LIN {X 0,Y 297.37,Z 514.484,A -85,B 0,C 180,E1 -16463.214,E2 -16463.214} C_VEL
LIN {X 0,Y 296.917,Z 516.954,A -85,B 0,C 180,E1 -16465.928,E2 -16465.928} C_VEL
LIN {X 0,Y 296.729,Z 518.18,A -85,B 0,C 180,E1 -16468.643,E2 -16468.643} C_VEL
LIN {X 0,Y 296.728,Z 518.204,A -85,B 0,C 180,E1 -16471.357,E2 -16471.357} C_VEL
LIN {X 0,Y 296.915,Z 517.029,A -85,B 0,C 180,E1 -16474.072,E2 -16474.072} C_VEL
LIN {X 0,Y 297.37,Z 514.612,A -85,B 0,C 180,E1 -16476.787,E2 -16476.787} C_VEL
LIN {X 0,Y 298.048,Z 510.874,A -85,B 0,C 180,E1 -16479.501,E2 -16479.501} C_VEL
LIN {X 0,Y 299.173,Z 505.674,A -85,B 0,C 180,E1 -16482.206,E2 -16482.206} C_VEL
LIN {X 0,Y 300.7,Z 498.834,A -85,B 0,C 180,E1 -16484.898,E2 -16484.898} C_VEL
LIN {X 0,Y 302.63,Z 491.286,A -85,B 0,C 180,E1 -16487.223,E2 -16487.223} C_VEL
LIN {X 0,Y 304.325,Z 483.451,A -85,B 0,C 180,E1 -16489.214,E2 -16489.214} C_VEL
LIN {X 0,Y 306.549,Z 474.009,A -85,B 0,C 180,E1 -16491.167,E2 -16491.167} C_VEL
LIN {X 0,Y 308.714,Z 463.565,A -85,B 0,C 180,E1 -16492.946,E2 -16492.946} C_VEL
LIN {X 0,Y 311.058,Z 452.04,A -85,B 0,C 180,E1 -16494.53,E2 -16494.53} C_VEL
LIN {X 0,Y 313.15,Z 439.163,A -85,B 0,C 180,E1 -16495.967,E2 -16495.967} C_VEL
LIN {X 0,Y 313.842,Z 434.12,A -85,B 0,C 180,E1 -16496.449,E2 -16496.449} C_VEL
LIN {X 0,Y 312.158,Z 424.12,A -85,B 0,C 180,E1 -16497.579,E2 -16497.579} C_VEL
LIN {X 0,Y 309.028,Z 411.527,A -85,B 0,C 180,E1 -16498.885,E2 -16498.885} C_VEL
LIN {X 0,Y 305.023,Z 398.954,A -85,B 0,C 180,E1 -16500.071,E2 -16500.071} C_VEL
LIN {X 0,Y 300.09,Z 386.492,A -85,B 0,C 180,E1 -16501.166,E2 -16501.166} C_VEL
LIN {X 0,Y 298.999,Z 383.235,A -85,B 0,C 180,E1 -16501.435,E2 -16501.435} C_VEL
LIN {X 0,Y 299.406,Z 379.396,A -85,B 0,C 180,E1 -16504.758,E2 -16504.758} C_VEL
LIN {X 0,Y 299.702,Z 376.329,A -85,B 0,C 180,E1 -16507.568,E2 -16507.568} C_VEL
LIN {X 0,Y 299.78,Z 374.508,A -85,B 0,C 180,E1 -16509.317,E2 -16509.317} C_VEL
LIN {X 0,Y 299.694,Z 372.408,A -85,B 0,C 180,E1 -16511.373,E2 -16511.373} C_VEL
LIN {X 0,Y 299.198,Z 368.796,A -85,B 0,C 180,E1 -16515.196,E2 -16515.196} C_VEL
LIN {X 0,Y 298.695,Z 365.599,A -85,B 0,C 180,E1 -16518.845,E2 -16518.845} C_VEL
LIN {X 0,Y 298.437,Z 363.932,A -85,B 0,C 180,E1 -16520.999,E2 -16520.999} C_VEL
LIN {X 0,Y 298.422,Z 363.937,A -85,B 0,C 180,E1 -16523.93,E2 -16523.93} C_VEL
LIN {X 0,Y 298.399,Z 363.939,A -85,B 0,C 180,E1 -16527.983,E2 -16527.983} C_VEL
LIN {X 0,Y 298.468,Z 363.93,A -85,B 0,C 180,E1 -16531.904,E2 -16531.904} C_VEL
LIN {X 0,Y 298.49,Z 363.929,A -85,B 0,C 180,E1 -16534.924,E2 -16534.924} C_VEL
LIN {X 0,Y 298.454,Z 363.928,A -85,B 0,C 180,E1 -16539.315,E2 -16539.315} C_VEL
LIN {X 0,Y 298.542,Z 363.918,A -85,B 0,C 180,E1 -16542.179,E2 -16542.179} C_VEL
LIN {X 0,Y 298.59,Z 363.912,A -85,B 0,C 180,E1 -16544.574,E2 -16544.574} C_VEL
LIN {X 0,Y 297.982,Z 363.99,A -85,B 0,C 180,E1 -16545.699,E2 -16545.699} C_VEL
LIN {X 0,Y 295.123,Z 364.351,A -85,B 0,C 180,E1 -16547.531,E2 -16547.531} C_VEL
LIN {X 0,Y 292.696,Z 364.654,A -85,B 0,C 180,E1 -16549.017,E2 -16549.017} C_VEL
LIN {X 0,Y 291.706,Z 364.774,A -85,B 0,C 180,E1 -16550.17,E2 -16550.17} C_VEL
LIN {X 0,Y 291.656,Z 364.777,A -85,B 0,C 180,E1 -16550.56,E2 -16550.56} C_VEL
LIN {X 0,Y 291.752,Z 364.769,A -85,B 0,C 180,E1 -16553.082,E2 -16553.082} C_VEL
LIN {X 0,Y 291.893,Z 364.745,A -85,B 0,C 180,E1 -16558.62,E2 -16558.62} C_VEL
LIN {X 0,Y 291.893,Z 364.745,A -85,B 0,C 180,E1 -16561.379,E2 -16561.379} C_VEL
LIN {X 0,Y 291.727,Z 364.771,A -85,B 0,C 180,E1 -16566.918,E2 -16566.918} C_VEL
LIN {X 0,Y 291.577,Z 364.793,A -85,B 0,C 180,E1 -16569.713,E2 -16569.713} C_VEL
LIN {X 0,Y 291.527,Z 364.795,A -85,B 0,C 180,E1 -16573.95,E2 -16573.95} C_VEL
LIN {X 0,Y 291.491,Z 364.802,A -85,B 0,C 180,E1 -16576.817,E2 -16576.817} C_VEL
LIN {X 0,Y 291.454,Z 364.806,A -85,B 0,C 180,E1 -16579.874,E2 -16579.874} C_VEL
LIN {X 0,Y 291.404,Z 364.815,A -85,B 0,C 180,E1 -16584.205,E2 -16584.205} C_VEL
LIN {X 0,Y 291.426,Z 364.81,A -85,B 0,C 180,E1 -16587.271,E2 -16587.271} C_VEL
LIN {X 0,Y 291.341,Z 364.818,A -85,B 0,C 180,E1 -16590.436,E2 -16590.436} C_VEL
LIN {X 0,Y 291.371,Z 364.967,A -85,B 0,C 180,E1 -16592.63,E2 -16592.63} C_VEL
LIN {X 0,Y 291.946,Z 367.659,A -85,B 0,C 180,E1 -16595.292,E2 -16595.292} C_VEL
LIN {X 0,Y 292.639,Z 371.276,A -85,B 0,C 180,E1 -16598.639,E2 -16598.639} C_VEL
LIN {X 0,Y 293.493,Z 375.469,A -85,B 0,C 180,E1 -16602.105,E2 -16602.105} C_VEL
LIN {X 0,Y 294.53,Z 380.83,A -85,B 0,C 180,E1 -16606.211,E2 -16606.211} C_VEL
LIN {X 0,Y 295.49,Z 386.215,A -85,B 0,C 180,E1 -16610.045,E2 -16610.045} C_VEL
LIN {X 0,Y 296.115,Z 390.267,A -85,B 0,C 180,E1 -16612.755,E2 -16612.755} C_VEL
LIN {X 0,Y 295.651,Z 393.125,A -85,B 0,C 180,E1 -16614.523,E2 -16614.523} C_VEL
LIN {X 0,Y 295.257,Z 394.696,A -85,B 0,C 180,E1 -16615.467,E2 -16615.467} C_VEL
LIN {X 0,Y 298.115,Z 404.031,A -85,B 0,C 180,E1 -16616.148,E2 -16616.148} C_VEL
LIN {X 0,Y 302.094,Z 419.344,A -85,B 0,C 180,E1 -16617.377,E2 -16617.377} C_VEL
LIN {X 0,Y 304.904,Z 434.204,A -85,B 0,C 180,E1 -16618.725,E2 -16618.725} C_VEL
LIN {X 0,Y 306.458,Z 447.084,A -85,B 0,C 180,E1 -16620.039,E2 -16620.039} C_VEL
LIN {X 0,Y 306.776,Z 452.763,A -85,B 0,C 180,E1 -16620.66,E2 -16620.66} C_VEL
LIN {X 0,Y 304.582,Z 465.397,A -85,B 0,C 180,E1 -16621.956,E2 -16621.956} C_VEL
LIN {X 0,Y 301.948,Z 478.242,A -85,B 0,C 180,E1 -16623.567,E2 -16623.567} C_VEL
LIN {X 0,Y 299.907,Z 488.037,A -85,B 0,C 180,E1 -16625.051,E2 -16625.051} C_VEL
LIN {X 0,Y 297.566,Z 498.682,A -85,B 0,C 180,E1 -16626.964,E2 -16626.964} C_VEL
LIN {X 0,Y 295.508,Z 508.524,A -85,B 0,C 180,E1 -16629.099,E2 -16629.099} C_VEL
LIN {X 0,Y 293.411,Z 517.704,A -85,B 0,C 180,E1 -16631.495,E2 -16631.495} C_VEL
LIN {X 0,Y 291.882,Z 525.537,A -85,B 0,C 180,E1 -16633.996,E2 -16633.996} C_VEL
LIN {X 0,Y 290.679,Z 532.426,A -85,B 0,C 180,E1 -16636.721,E2 -16636.721} C_VEL
LIN {X 0,Y 289.903,Z 537.976,A -85,B 0,C 180,E1 -16639.524,E2 -16639.524} C_VEL
LIN {X 0,Y 289.637,Z 541.184,A -85,B 0,C 180,E1 -16641.628,E2 -16641.628} C_VEL
LIN {X 0,Y 289.515,Z 544.352,A -85,B 0,C 180,E1 -16644.428,E2 -16644.428} C_VEL
LIN {X 0,Y 289.519,Z 546.244,A -85,B 0,C 180,E1 -16647.217,E2 -16647.217} C_VEL
LIN {X 0,Y 289.58,Z 546.886,A -85,B 0,C 180,E1 -16650,E2 -16650} C_VEL
LIN {X 0,Y 289.522,Z 546.235,A -85,B 0,C 180,E1 -16652.783,E2 -16652.783} C_VEL
LIN {X 0,Y 289.55,Z 544.272,A -85,B 0,C 180,E1 -16655.642,E2 -16655.642} C_VEL
LIN {X 0,Y 289.637,Z 541.156,A -85,B 0,C 180,E1 -16658.371,E2 -16658.371} C_VEL
LIN {X 0,Y 290.02,Z 536.65,A -85,B 0,C 180,E1 -16661.178,E2 -16661.178} C_VEL
LIN {X 0,Y 290.906,Z 530.713,A -85,B 0,C 180,E1 -16663.98,E2 -16663.98} C_VEL
LIN {X 0,Y 292.297,Z 523.193,A -85,B 0,C 180,E1 -16666.77,E2 -16666.77} C_VEL
LIN {X 0,Y 293.903,Z 515.126,A -85,B 0,C 180,E1 -16669.196,E2 -16669.196} C_VEL
LIN {X 0,Y 296.092,Z 505.429,A -85,B 0,C 180,E1 -16671.587,E2 -16671.587} C_VEL
LIN {X 0,Y 298.214,Z 495.509,A -85,B 0,C 180,E1 -16673.618,E2 -16673.618} C_VEL
LIN {X 0,Y 300.741,Z 483.712,A -85,B 0,C 180,E1 -16675.615,E2 -16675.615} C_VEL
LIN {X 0,Y 303.171,Z 471.961,A -85,B 0,C 180,E1 -16677.248,E2 -16677.248} C_VEL
LIN {X 0,Y 305.675,Z 459.264,A -85,B 0,C 180,E1 -16678.682,E2 -16678.682} C_VEL
LIN {X 0,Y 306.763,Z 451.271,A -85,B 0,C 180,E1 -16679.474,E2 -16679.474} C_VEL
LIN {X 0,Y 305.283,Z 437.149,A -85,B 0,C 180,E1 -16680.959,E2 -16680.959} C_VEL
LIN {X 0,Y 302.891,Z 423.088,A -85,B 0,C 180,E1 -16682.264,E2 -16682.264} C_VEL
LIN {X 0,Y 299.26,Z 408.308,A -85,B 0,C 180,E1 -16683.495,E2 -16683.495} C_VEL
LIN {X 0,Y 295.225,Z 394.702,A -85,B 0,C 180,E1 -16684.5,E2 -16684.5} C_VEL
LIN {X 0,Y 295.95,Z 391.521,A -85,B 0,C 180,E1 -16686.419,E2 -16686.419} C_VEL
LIN {X 0,Y 295.895,Z 388.478,A -85,B 0,C 180,E1 -16688.39,E2 -16688.39} C_VEL
LIN {X 0,Y 294.873,Z 382.73,A -85,B 0,C 180,E1 -16692.367,E2 -16692.367} C_VEL
LIN {X 0,Y 293.937,Z 377.696,A -85,B 0,C 180,E1 -16696.102,E2 -16696.102} C_VEL
LIN {X 0,Y 293.069,Z 373.272,A -85,B 0,C 180,E1 -16699.648,E2 -16699.648} C_VEL
LIN {X 0,Y 292.307,Z 369.354,A -85,B 0,C 180,E1 -16703.053,E2 -16703.053} C_VEL
LIN {X 0,Y 291.425,Z 365.233,A -85,B 0,C 180,E1 -16707.024,E2 -16707.024} C_VEL
LIN {X 0,Y 291.346,Z 364.824,A -85,B 0,C 180,E1 -16707.596,E2 -16707.596} C_VEL
LIN {X 0,Y 291.387,Z 364.819,A -85,B 0,C 180,E1 -16711.159,E2 -16711.159} C_VEL
LIN {X 0,Y 291.422,Z 364.808,A -85,B 0,C 180,E1 -16714.273,E2 -16714.273} C_VEL
LIN {X 0,Y 291.384,Z 364.814,A -85,B 0,C 180,E1 -16717.3,E2 -16717.3} C_VEL
LIN {X 0,Y 291.46,Z 364.804,A -85,B 0,C 180,E1 -16720.271,E2 -16720.271} C_VEL
LIN {X 0,Y 291.557,Z 364.786,A -85,B 0,C 180,E1 -16724.624,E2 -16724.624} C_VEL
LIN {X 0,Y 291.54,Z 364.795,A -85,B 0,C 180,E1 -16728.881,E2 -16728.881} C_VEL
LIN {X 0,Y 291.671,Z 364.78,A -85,B 0,C 180,E1 -16731.688,E2 -16731.688} C_VEL
LIN {X 0,Y 291.628,Z 364.78,A -85,B 0,C 180,E1 -16734.469,E2 -16734.469} C_VEL
LIN {X 0,Y 291.893,Z 364.752,A -85,B 0,C 180,E1 -16738.621,E2 -16738.621} C_VEL
LIN {X 0,Y 291.892,Z 364.745,A -85,B 0,C 180,E1 -16741.38,E2 -16741.38} C_VEL
LIN {X 0,Y 291.75,Z 364.765,A -85,B 0,C 180,E1 -16746.918,E2 -16746.918} C_VEL
LIN {X 0,Y 291.633,Z 364.785,A -85,B 0,C 180,E1 -16749.712,E2 -16749.712} C_VEL
LIN {X 0,Y 291.527,Z 364.794,A -85,B 0,C 180,E1 -16753.95,E2 -16753.95} C_VEL
LIN {X 0,Y 291.491,Z 364.801,A -85,B 0,C 180,E1 -16756.818,E2 -16756.818} C_VEL
LIN {X 0,Y 291.453,Z 364.808,A -85,B 0,C 180,E1 -16759.875,E2 -16759.875} C_VEL
LIN {X 0,Y 291.403,Z 364.805,A -85,B 0,C 180,E1 -16764.205,E2 -16764.205} C_VEL
LIN {X 0,Y 291.425,Z 364.804,A -85,B 0,C 180,E1 -16767.272,E2 -16767.272} C_VEL
LIN {X 0,Y 291.34,Z 364.818,A -85,B 0,C 180,E1 -16770.437,E2 -16770.437} C_VEL
LIN {X 0,Y 291.347,Z 364.819,A -85,B 0,C 180,E1 -16773.698,E2 -16773.698} C_VEL
LIN {X 0,Y 291.375,Z 364.817,A -85,B 0,C 180,E1 -16777.253,E2 -16777.253} C_VEL
LIN {X 0,Y 291.385,Z 364.97,A -85,B 0,C 180,E1 -16778.622,E2 -16778.622} C_VEL
LIN {X 0,Y 291.885,Z 368.062,A -85,B 0,C 180,E1 -16782.391,E2 -16782.391} C_VEL
LIN {X 0,Y 292.435,Z 371.328,A -85,B 0,C 180,E1 -16786.136,E2 -16786.136} C_VEL
LIN {X 0,Y 292.753,Z 374.6,A -85,B 0,C 180,E1 -16789.595,E2 -16789.595} C_VEL
LIN {X 0,Y 292.644,Z 378.189,A -85,B 0,C 180,E1 -16793.102,E2 -16793.102} C_VEL
LIN {X 0,Y 292.223,Z 381.859,A -85,B 0,C 180,E1 -16796.416,E2 -16796.416} C_VEL
LIN {X 0,Y 292.078,Z 383.466,A -85,B 0,C 180,E1 -16797.834,E2 -16797.834} C_VEL
LIN {X 0,Y 293.241,Z 386.749,A -85,B 0,C 180,E1 -16798.103,E2 -16798.103} C_VEL
LIN {X 0,Y 298.534,Z 400.073,A -85,B 0,C 180,E1 -16799.335,E2 -16799.335} C_VEL
LIN {X 0,Y 302.565,Z 412.598,A -85,B 0,C 180,E1 -16800.583,E2 -16800.583} C_VEL
LIN {X 0,Y 305.59,Z 425.125,A -85,B 0,C 180,E1 -16801.933,E2 -16801.933} C_VEL
LIN {X 0,Y 307.35,Z 434.992,A -85,B 0,C 180,E1 -16803.1,E2 -16803.1} C_VEL
LIN {X 0,Y 305.683,Z 446.293,A -85,B 0,C 180,E1 -16804.281,E2 -16804.281} C_VEL
LIN {X 0,Y 303.559,Z 457.781,A -85,B 0,C 180,E1 -16805.736,E2 -16805.736} C_VEL
LIN {X 0,Y 301.21,Z 468.343,A -85,B 0,C 180,E1 -16807.357,E2 -16807.357} C_VEL
LIN {X 0,Y 298.819,Z 478.827,A -85,B 0,C 180,E1 -16809.342,E2 -16809.342} C_VEL
LIN {X 0,Y 296.706,Z 487.48,A -85,B 0,C 180,E1 -16811.347,E2 -16811.347} C_VEL
LIN {X 0,Y 294.766,Z 495.809,A -85,B 0,C 180,E1 -16813.731,E2 -16813.731} C_VEL
LIN {X 0,Y 293.031,Z 502.541,A -85,B 0,C 180,E1 -16816.123,E2 -16816.123} C_VEL
LIN {X 0,Y 291.594,Z 508.601,A -85,B 0,C 180,E1 -16818.883,E2 -16818.883} C_VEL
LIN {X 0,Y 290.647,Z 513.109,A -85,B 0,C 180,E1 -16821.658,E2 -16821.658} C_VEL
LIN {X 0,Y 290.078,Z 516.224,A -85,B 0,C 180,E1 -16824.439,E2 -16824.439} C_VEL
LIN {X 0,Y 289.712,Z 518.065,A -85,B 0,C 180,E1 -16827.219,E2 -16827.219} C_VEL
LIN {X 0,Y 289.594,Z 518.687,A -85,B 0,C 180,E1 -16830,E2 -16830} C_VEL
LIN {X 0,Y 289.711,Z 518.113,A -85,B 0,C 180,E1 -16832.781,E2 -16832.781} C_VEL
LIN {X 0,Y 290.059,Z 516.324,A -85,B 0,C 180,E1 -16835.562,E2 -16835.562} C_VEL
LIN {X 0,Y 290.645,Z 513.261,A -85,B 0,C 180,E1 -16838.342,E2 -16838.342} C_VEL
LIN {X 0,Y 291.572,Z 508.818,A -85,B 0,C 180,E1 -16841.118,E2 -16841.118} C_VEL
LIN {X 0,Y 292.952,Z 502.829,A -85,B 0,C 180,E1 -16843.881,E2 -16843.881} C_VEL
LIN {X 0,Y 294.741,Z 496.162,A -85,B 0,C 180,E1 -16846.271,E2 -16846.271} C_VEL
LIN {X 0,Y 296.503,Z 488.39,A -85,B 0,C 180,E1 -16848.536,E2 -16848.536} C_VEL
LIN {X 0,Y 298.705,Z 479.34,A -85,B 0,C 180,E1 -16850.667,E2 -16850.667} C_VEL
LIN {X 0,Y 301.136,Z 468.954,A -85,B 0,C 180,E1 -16852.649,E2 -16852.649} C_VEL
LIN {X 0,Y 303.481,Z 458.512,A -85,B 0,C 180,E1 -16854.271,E2 -16854.271} C_VEL
LIN {X 0,Y 305.566,Z 447.194,A -85,B 0,C 180,E1 -16855.73,E2 -16855.73} C_VEL
LIN {X 0,Y 307.42,Z 435.802,A -85,B 0,C 180,E1 -16856.926,E2 -16856.926} C_VEL
LIN {X 0,Y 305.267,Z 423.348,A -85,B 0,C 180,E1 -16858.384,E2 -16858.384} C_VEL
LIN {X 0,Y 301.631,Z 409.433,A -85,B 0,C 180,E1 -16859.864,E2 -16859.864} C_VEL
LIN {X 0,Y 297.328,Z 396.7,A -85,B 0,C 180,E1 -16861.109,E2 -16861.109} C_VEL
LIN {X 0,Y 292.847,Z 385.944,A -85,B 0,C 180,E1 -16862.097,E2 -16862.097} C_VEL
LIN {X 0,Y 292.067,Z 383.454,A -85,B 0,C 180,E1 -16862.302,E2 -16862.302} C_VEL
LIN {X 0,Y 292.445,Z 380.152,A -85,B 0,C 180,E1 -16865.224,E2 -16865.224} C_VEL
LIN {X 0,Y 292.764,Z 376.571,A -85,B 0,C 180,E1 -16868.62,E2 -16868.62} C_VEL
LIN {X 0,Y 292.651,Z 373.314,A -85,B 0,C 180,E1 -16871.887,E2 -16871.887} C_VEL
LIN {X 0,Y 292.163,Z 369.759,A -85,B 0,C 180,E1 -16875.765,E2 -16875.765} C_VEL
LIN {X 0,Y 291.685,Z 366.668,A -85,B 0,C 180,E1 -16879.416,E2 -16879.416} C_VEL
LIN {X 0,Y 291.371,Z 364.813,A -85,B 0,C 180,E1 -16881.803,E2 -16881.803} C_VEL
LIN {X 0,Y 291.373,Z 364.817,A -85,B 0,C 180,E1 -16885.095,E2 -16885.095} C_VEL
LIN {X 0,Y 291.376,Z 364.814,A -85,B 0,C 180,E1 -16887.951,E2 -16887.951} C_VEL
LIN {X 0,Y 291.386,Z 364.813,A -85,B 0,C 180,E1 -16891.159,E2 -16891.159} C_VEL
LIN {X 0,Y 291.421,Z 364.806,A -85,B 0,C 180,E1 -16894.272,E2 -16894.272} C_VEL
LIN {X 0,Y 291.386,Z 364.814,A -85,B 0,C 180,E1 -16897.3,E2 -16897.3} C_VEL
LIN {X 0,Y 291.462,Z 364.806,A -85,B 0,C 180,E1 -16900.27,E2 -16900.27} C_VEL
LIN {X 0,Y 291.559,Z 364.788,A -85,B 0,C 180,E1 -16904.624,E2 -16904.624} C_VEL
LIN {X 0,Y 291.542,Z 364.791,A -85,B 0,C 180,E1 -16908.881,E2 -16908.881} C_VEL
LIN {X 0,Y 291.656,Z 364.777,A -85,B 0,C 180,E1 -16910.56,E2 -16910.56} C_VEL
LIN {X 0,Y 291.383,Z 364.809,A -85,B 0,C 180,E1 -16911.331,E2 -16911.331} C_VEL
LIN {X 0,Y 290.021,Z 364.983,A -85,B 0,C 180,E1 -16912.468,E2 -16912.468} C_VEL
LIN {X 0,Y 285.621,Z 365.529,A -85,B 0,C 180,E1 -16915.111,E2 -16915.111} C_VEL
LIN {X 0,Y 284.668,Z 365.651,A -85,B 0,C 180,E1 -16916.294,E2 -16916.294} C_VEL
LIN {X 0,Y 284.65,Z 365.649,A -85,B 0,C 180,E1 -16916.694,E2 -16916.694} C_VEL
LIN {X 0,Y 284.928,Z 365.62,A -85,B 0,C 180,E1 -16920,E2 -16920} C_VEL
LIN {X 0,Y 284.747,Z 365.641,A -85,B 0,C 180,E1 -16922.829,E2 -16922.829} C_VEL
LIN {X 0,Y 284.678,Z 365.647,A -85,B 0,C 180,E1 -16927.09,E2 -16927.09} C_VEL
LIN {X 0,Y 284.522,Z 365.671,A -85,B 0,C 180,E1 -16929.957,E2 -16929.957} C_VEL
LIN {X 0,Y 284.487,Z 365.673,A -85,B 0,C 180,E1 -16934.302,E2 -16934.302} C_VEL
LIN {X 0,Y 284.43,Z 365.681,A -85,B 0,C 180,E1 -16937.248,E2 -16937.248} C_VEL
LIN {X 0,Y 284.384,Z 365.687,A -85,B 0,C 180,E1 -16940.242,E2 -16940.242} C_VEL
LIN {X 0,Y 284.373,Z 365.692,A -85,B 0,C 180,E1 -16943.875,E2 -16943.875} C_VEL
LIN {X 0,Y 284.4,Z 365.685,A -85,B 0,C 180,E1 -16947.173,E2 -16947.173} C_VEL
LIN {X 0,Y 284.299,Z 365.7,A -85,B 0,C 180,E1 -16951.274,E2 -16951.274} C_VEL
LIN {X 0,Y 284.976,Z 368.813,A -85,B 0,C 180,E1 -16954.556,E2 -16954.556} C_VEL
LIN {X 0,Y 285.691,Z 372.513,A -85,B 0,C 180,E1 -16958.075,E2 -16958.075} C_VEL
LIN {X 0,Y 286.476,Z 376.426,A -85,B 0,C 180,E1 -16961.481,E2 -16961.481} C_VEL
LIN {X 0,Y 287.348,Z 381.061,A -85,B 0,C 180,E1 -16965.177,E2 -16965.177} C_VEL
LIN {X 0,Y 288.301,Z 386.346,A -85,B 0,C 180,E1 -16969.086,E2 -16969.086} C_VEL
LIN {X 0,Y 289.102,Z 391.33,A -85,B 0,C 180,E1 -16972.573,E2 -16972.573} C_VEL
LIN {X 0,Y 288.719,Z 393.944,A -85,B 0,C 180,E1 -16974.252,E2 -16974.252} C_VEL
LIN {X 0,Y 288.568,Z 394.496,A -85,B 0,C 180,E1 -16974.592,E2 -16974.592} C_VEL
LIN {X 0,Y 291.432,Z 403.799,A -85,B 0,C 180,E1 -16975.305,E2 -16975.305} C_VEL
LIN {X 0,Y 295.43,Z 418.879,A -85,B 0,C 180,E1 -16976.571,E2 -16976.571} C_VEL
LIN {X 0,Y 298.17,Z 432.949,A -85,B 0,C 180,E1 -16977.893,E2 -16977.893} C_VEL
LIN {X 0,Y 299.659,Z 444.735,A -85,B 0,C 180,E1 -16979.117,E2 -16979.117} C_VEL
LIN {X 0,Y 300.331,Z 453.325,A -85,B 0,C 180,E1 -16980.086,E2 -16980.086} C_VEL
LIN {X 0,Y 298.011,Z 466.352,A -85,B 0,C 180,E1 -16981.474,E2 -16981.474} C_VEL
LIN {X 0,Y 295.292,Z 478.986,A -85,B 0,C 180,E1 -16983.114,E2 -16983.114} C_VEL
LIN {X 0,Y 292.964,Z 489.599,A -85,B 0,C 180,E1 -16984.798,E2 -16984.798} C_VEL
LIN {X 0,Y 290.514,Z 500.257,A -85,B 0,C 180,E1 -16986.821,E2 -16986.821} C_VEL
LIN {X 0,Y 288.159,Z 510.909,A -85,B 0,C 180,E1 -16989.289,E2 -16989.289} C_VEL
LIN {X 0,Y 286.088,Z 519.627,A -85,B 0,C 180,E1 -16991.747,E2 -16991.747} C_VEL
LIN {X 0,Y 284.566,Z 527.296,A -85,B 0,C 180,E1 -16994.405,E2 -16994.405} C_VEL
LIN {X 0,Y 283.457,Z 533.558,A -85,B 0,C 180,E1 -16997.106,E2 -16997.106} C_VEL
LIN {X 0,Y 282.725,Z 538.754,A -85,B 0,C 180,E1 -16999.979,E2 -16999.979} C_VEL
LIN {X 0,Y 282.466,Z 542.582,A -85,B 0,C 180,E1 -17002.853,E2 -17002.853} C_VEL
LIN {X 0,Y 282.411,Z 545.109,A -85,B 0,C 180,E1 -17005.718,E2 -17005.718} C_VEL
LIN {X 0,Y 282.446,Z 546.378,A -85,B 0,C 180,E1 -17008.574,E2 -17008.574} C_VEL
LIN {X 0,Y 282.493,Z 546.541,A -85,B 0,C 180,E1 -17010,E2 -17010} C_VEL
LIN {X 0,Y 282.448,Z 545.89,A -85,B 0,C 180,E1 -17012.852,E2 -17012.852} C_VEL
LIN {X 0,Y 282.463,Z 543.984,A -85,B 0,C 180,E1 -17015.712,E2 -17015.712} C_VEL
LIN {X 0,Y 282.575,Z 540.805,A -85,B 0,C 180,E1 -17018.582,E2 -17018.582} C_VEL
LIN {X 0,Y 282.987,Z 536.295,A -85,B 0,C 180,E1 -17021.46,E2 -17021.46} C_VEL
LIN {X 0,Y 283.944,Z 530.354,A -85,B 0,C 180,E1 -17024.33,E2 -17024.33} C_VEL
LIN {X 0,Y 285.422,Z 522.828,A -85,B 0,C 180,E1 -17027.186,E2 -17027.186} C_VEL
LIN {X 0,Y 287.112,Z 514.751,A -85,B 0,C 180,E1 -17029.668,E2 -17029.668} C_VEL
LIN {X 0,Y 289.394,Z 505.041,A -85,B 0,C 180,E1 -17032.112,E2 -17032.112} C_VEL
LIN {X 0,Y 291.639,Z 495.106,A -85,B 0,C 180,E1 -17034.184,E2 -17034.184} C_VEL
LIN {X 0,Y 294.279,Z 483.286,A -85,B 0,C 180,E1 -17036.22,E2 -17036.22} C_VEL
LIN {X 0,Y 296.797,Z 471.503,A -85,B 0,C 180,E1 -17037.883,E2 -17037.883} C_VEL
LIN {X 0,Y 299.432,Z 458.763,A -85,B 0,C 180,E1 -17039.338,E2 -17039.338} C_VEL
LIN {X 0,Y 300.265,Z 452.33,A -85,B 0,C 180,E1 -17040.001,E2 -17040.001} C_VEL
LIN {X 0,Y 298.95,Z 438.724,A -85,B 0,C 180,E1 -17041.496,E2 -17041.496} C_VEL
LIN {X 0,Y 296.619,Z 424.538,A -85,B 0,C 180,E1 -17042.883,E2 -17042.883} C_VEL
LIN {X 0,Y 293.229,Z 410.18,A -85,B 0,C 180,E1 -17044.144,E2 -17044.144} C_VEL
LIN {X 0,Y 288.548,Z 394.468,A -85,B 0,C 180,E1 -17045.393,E2 -17045.393} C_VEL
LIN {X 0,Y 289.073,Z 391.269,A -85,B 0,C 180,E1 -17047.431,E2 -17047.431} C_VEL
LIN {X 0,Y 288.499,Z 387.445,A -85,B 0,C 180,E1 -17050.08,E2 -17050.08} C_VEL
LIN {X 0,Y 287.553,Z 382.09,A -85,B 0,C 180,E1 -17053.99,E2 -17053.99} C_VEL
LIN {X 0,Y 286.737,Z 377.831,A -85,B 0,C 180,E1 -17057.334,E2 -17057.334} C_VEL
LIN {X 0,Y 286.042,Z 374.282,A -85,B 0,C 180,E1 -17060.297,E2 -17060.297} C_VEL
LIN {X 0,Y 285.15,Z 369.758,A -85,B 0,C 180,E1 -17064.424,E2 -17064.424} C_VEL
LIN {X 0,Y 284.304,Z 365.7,A -85,B 0,C 180,E1 -17068.649,E2 -17068.649} C_VEL
LIN {X 0,Y 284.401,Z 365.685,A -85,B 0,C 180,E1 -17072.826,E2 -17072.826} C_VEL
LIN {X 0,Y 284.369,Z 365.685,A -85,B 0,C 180,E1 -17076.707,E2 -17076.707} C_VEL
LIN {X 0,Y 284.406,Z 365.678,A -85,B 0,C 180,E1 -17081.262,E2 -17081.262} C_VEL
LIN {X 0,Y 284.494,Z 365.665,A -85,B 0,C 180,E1 -17084.459,E2 -17084.459} C_VEL
LIN {X 0,Y 284.491,Z 365.674,A -85,B 0,C 180,E1 -17088.602,E2 -17088.602} C_VEL
LIN {X 0,Y 284.625,Z 365.655,A -85,B 0,C 180,E1 -17091.48,E2 -17091.48} C_VEL
LIN {X 0,Y 284.597,Z 365.655,A -85,B 0,C 180,E1 -17094.331,E2 -17094.331} C_VEL
LIN {X 0,Y 284.859,Z 365.629,A -85,B 0,C 180,E1 -17098.587,E2 -17098.587} C_VEL
LIN {X 0,Y 284.858,Z 365.621,A -85,B 0,C 180,E1 -17101.414,E2 -17101.414} C_VEL
LIN {X 0,Y 284.702,Z 365.642,A -85,B 0,C 180,E1 -17107.09,E2 -17107.09} C_VEL
LIN {X 0,Y 284.57,Z 365.664,A -85,B 0,C 180,E1 -17109.955,E2 -17109.955} C_VEL
LIN {X 0,Y 284.486,Z 365.669,A -85,B 0,C 180,E1 -17114.303,E2 -17114.303} C_VEL
LIN {X 0,Y 284.429,Z 365.679,A -85,B 0,C 180,E1 -17117.248,E2 -17117.248} C_VEL
LIN {X 0,Y 284.381,Z 365.685,A -85,B 0,C 180,E1 -17120.242,E2 -17120.242} C_VEL
LIN {X 0,Y 284.372,Z 365.682,A -85,B 0,C 180,E1 -17123.876,E2 -17123.876} C_VEL
LIN {X 0,Y 284.4,Z 365.679,A -85,B 0,C 180,E1 -17127.174,E2 -17127.174} C_VEL
LIN {X 0,Y 284.299,Z 365.697,A -85,B 0,C 180,E1 -17131.274,E2 -17131.274} C_VEL
LIN {X 0,Y 284.343,Z 365.693,A -85,B 0,C 180,E1 -17135.348,E2 -17135.348} C_VEL
LIN {X 0,Y 284.359,Z 365.878,A -85,B 0,C 180,E1 -17137.731,E2 -17137.731} C_VEL
LIN {X 0,Y 284.892,Z 369.049,A -85,B 0,C 180,E1 -17141.764,E2 -17141.764} C_VEL
LIN {X 0,Y 285.405,Z 372.268,A -85,B 0,C 180,E1 -17145.571,E2 -17145.571} C_VEL
LIN {X 0,Y 285.729,Z 374.826,A -85,B 0,C 180,E1 -17148.386,E2 -17148.386} C_VEL
LIN {X 0,Y 285.793,Z 376.621,A -85,B 0,C 180,E1 -17150.255,E2 -17150.255} C_VEL
LIN {X 0,Y 285.737,Z 378.426,A -85,B 0,C 180,E1 -17152.055,E2 -17152.055} C_VEL
LIN {X 0,Y 285.332,Z 382.107,A -85,B 0,C 180,E1 -17155.492,E2 -17155.492} C_VEL
LIN {X 0,Y 285.17,Z 383.727,A -85,B 0,C 180,E1 -17156.923,E2 -17156.923} C_VEL
LIN {X 0,Y 286.3,Z 386.895,A -85,B 0,C 180,E1 -17157.186,E2 -17157.186} C_VEL
LIN {X 0,Y 291.115,Z 398.564,A -85,B 0,C 180,E1 -17158.323,E2 -17158.323} C_VEL
LIN {X 0,Y 295.605,Z 411.983,A -85,B 0,C 180,E1 -17159.714,E2 -17159.714} C_VEL
LIN {X 0,Y 298.79,Z 424.625,A -85,B 0,C 180,E1 -17161.126,E2 -17161.126} C_VEL
LIN {X 0,Y 300.967,Z 437.063,A -85,B 0,C 180,E1 -17162.652,E2 -17162.652} C_VEL
LIN {X 0,Y 298.826,Z 449.547,A -85,B 0,C 180,E1 -17164.021,E2 -17164.021} C_VEL
LIN {X 0,Y 296.325,Z 461.601,A -85,B 0,C 180,E1 -17165.664,E2 -17165.664} C_VEL
LIN {X 0,Y 294.29,Z 470.683,A -85,B 0,C 180,E1 -17167.165,E2 -17167.165} C_VEL
LIN {X 0,Y 291.803,Z 480.808,A -85,B 0,C 180,E1 -17169.191,E2 -17169.191} C_VEL
LIN {X 0,Y 289.703,Z 488.943,A -85,B 0,C 180,E1 -17171.18,E2 -17171.18} C_VEL
LIN {X 0,Y 287.671,Z 497.254,A -85,B 0,C 180,E1 -17173.683,E2 -17173.683} C_VEL
LIN {X 0,Y 286.12,Z 502.899,A -85,B 0,C 180,E1 -17175.781,E2 -17175.781} C_VEL
LIN {X 0,Y 284.618,Z 508.954,A -85,B 0,C 180,E1 -17178.607,E2 -17178.607} C_VEL
LIN {X 0,Y 283.616,Z 513.458,A -85,B 0,C 180,E1 -17181.45,E2 -17181.45} C_VEL
LIN {X 0,Y 283.019,Z 516.57,A -85,B 0,C 180,E1 -17184.3,E2 -17184.3} C_VEL
LIN {X 0,Y 282.638,Z 518.41,A -85,B 0,C 180,E1 -17187.15,E2 -17187.15} C_VEL
LIN {X 0,Y 282.508,Z 519.032,A -85,B 0,C 180,E1 -17190,E2 -17190} C_VEL
LIN {X 0,Y 282.637,Z 518.457,A -85,B 0,C 180,E1 -17192.851,E2 -17192.851} C_VEL
LIN {X 0,Y 283.003,Z 516.669,A -85,B 0,C 180,E1 -17195.701,E2 -17195.701} C_VEL
LIN {X 0,Y 283.612,Z 513.608,A -85,B 0,C 180,E1 -17198.551,E2 -17198.551} C_VEL
LIN {X 0,Y 284.599,Z 509.168,A -85,B 0,C 180,E1 -17201.394,E2 -17201.394} C_VEL
LIN {X 0,Y 286.044,Z 503.184,A -85,B 0,C 180,E1 -17204.223,E2 -17204.223} C_VEL
LIN {X 0,Y 287.937,Z 496.522,A -85,B 0,C 180,E1 -17206.666,E2 -17206.666} C_VEL
LIN {X 0,Y 289.69,Z 489.129,A -85,B 0,C 180,E1 -17208.887,E2 -17208.887} C_VEL
LIN {X 0,Y 292.095,Z 479.722,A -85,B 0,C 180,E1 -17211.156,E2 -17211.156} C_VEL
LIN {X 0,Y 294.608,Z 469.356,A -85,B 0,C 180,E1 -17213.18,E2 -17213.18} C_VEL
LIN {X 0,Y 297.035,Z 458.94,A -85,B 0,C 180,E1 -17214.833,E2 -17214.833} C_VEL
LIN {X 0,Y 299.216,Z 447.659,A -85,B 0,C 180,E1 -17216.317,E2 -17216.317} C_VEL
LIN {X 0,Y 300.993,Z 437.048,A -85,B 0,C 180,E1 -17217.466,E2 -17217.466} C_VEL
LIN {X 0,Y 298.791,Z 424.446,A -85,B 0,C 180,E1 -17219.011,E2 -17219.011} C_VEL
LIN {X 0,Y 295.515,Z 411.619,A -85,B 0,C 180,E1 -17220.445,E2 -17220.445} C_VEL
LIN {X 0,Y 290.891,Z 397.772,A -85,B 0,C 180,E1 -17221.873,E2 -17221.873} C_VEL
LIN {X 0,Y 286.329,Z 386.933,A -85,B 0,C 180,E1 -17222.935,E2 -17222.935} C_VEL
LIN {X 0,Y 285.281,Z 384.242,A -85,B 0,C 180,E1 -17223.171,E2 -17223.171} C_VEL
LIN {X 0,Y 285.177,Z 383.615,A -85,B 0,C 180,E1 -17223.247,E2 -17223.247} C_VEL
LIN {X 0,Y 285.564,Z 380.386,A -85,B 0,C 180,E1 -17226.205,E2 -17226.205} C_VEL
LIN {X 0,Y 285.751,Z 378.442,A -85,B 0,C 180,E1 -17228.09,E2 -17228.09} C_VEL
LIN {X 0,Y 285.806,Z 376.206,A -85,B 0,C 180,E1 -17230.333,E2 -17230.333} C_VEL
LIN {X 0,Y 285.494,Z 373.191,A -85,B 0,C 180,E1 -17233.574,E2 -17233.574} C_VEL
LIN {X 0,Y 284.97,Z 369.611,A -85,B 0,C 180,E1 -17237.721,E2 -17237.721} C_VEL
LIN {X 0,Y 284.688,Z 367.683,A -85,B 0,C 180,E1 -17240.069,E2 -17240.069} C_VEL
LIN {X 0,Y 284.371,Z 365.686,A -85,B 0,C 180,E1 -17242.944,E2 -17242.944} C_VEL
LIN {X 0,Y 284.312,Z 365.695,A -85,B 0,C 180,E1 -17247.19,E2 -17247.19} C_VEL
LIN {X 0,Y 284.363,Z 365.69,A -85,B 0,C 180,E1 -17250.376,E2 -17250.376} C_VEL
LIN {X 0,Y 284.382,Z 365.683,A -85,B 0,C 180,E1 -17253.587,E2 -17253.587} C_VEL
LIN {X 0,Y 284.371,Z 365.684,A -85,B 0,C 180,E1 -17256.707,E2 -17256.707} C_VEL
LIN {X 0,Y 284.408,Z 365.681,A -85,B 0,C 180,E1 -17261.262,E2 -17261.262} C_VEL
LIN {X 0,Y 284.497,Z 365.669,A -85,B 0,C 180,E1 -17264.459,E2 -17264.459} C_VEL
LIN {X 0,Y 284.493,Z 365.667,A -85,B 0,C 180,E1 -17268.601,E2 -17268.601} C_VEL
LIN {X 0,Y 284.664,Z 365.645,A -85,B 0,C 180,E1 -17271.481,E2 -17271.481} C_VEL
LIN {X 0,Y 284.606,Z 365.653,A -85,B 0,C 180,E1 -17274.331,E2 -17274.331} C_VEL
LIN {X 0,Y 284.65,Z 365.649,A -85,B 0,C 180,E1 -17276.694,E2 -17276.694} C_VEL
LIN {X 0,Y 284.179,Z 365.712,A -85,B 0,C 180,E1 -17277.877,E2 -17277.877} C_VEL
LIN {X 0,Y 282.734,Z 365.898,A -85,B 0,C 180,E1 -17279.04,E2 -17279.04} C_VEL
LIN {X 0,Y 278.139,Z 366.47,A -85,B 0,C 180,E1 -17282.174,E2 -17282.174} C_VEL
LIN {X 0,Y 277.682,Z 366.52,A -85,B 0,C 180,E1 -17282.994,E2 -17282.994} C_VEL
LIN {X 0,Y 277.632,Z 366.524,A -85,B 0,C 180,E1 -17287.271,E2 -17287.271} C_VEL
LIN {X 0,Y 277.465,Z 366.547,A -85,B 0,C 180,E1 -17290.213,E2 -17290.213} C_VEL
LIN {X 0,Y 277.439,Z 366.552,A -85,B 0,C 180,E1 -17294.674,E2 -17294.674} C_VEL
LIN {X 0,Y 277.35,Z 366.565,A -85,B 0,C 180,E1 -17299.233,E2 -17299.233} C_VEL
LIN {X 0,Y 277.332,Z 366.569,A -85,B 0,C 180,E1 -17303.92,E2 -17303.92} C_VEL
LIN {X 0,Y 277.329,Z 366.567,A -85,B 0,C 180,E1 -17307.505,E2 -17307.505} C_VEL
LIN {X 0,Y 277.307,Z 366.679,A -85,B 0,C 180,E1 -17310.186,E2 -17310.186} C_VEL
LIN {X 0,Y 277.941,Z 369.968,A -85,B 0,C 180,E1 -17313.799,E2 -17313.799} C_VEL
LIN {X 0,Y 278.656,Z 373.488,A -85,B 0,C 180,E1 -17317.251,E2 -17317.251} C_VEL
LIN {X 0,Y 279.49,Z 377.632,A -85,B 0,C 180,E1 -17321.029,E2 -17321.029} C_VEL
LIN {X 0,Y 280.501,Z 383.019,A -85,B 0,C 180,E1 -17325.448,E2 -17325.448} C_VEL
LIN {X 0,Y 281.466,Z 388.399,A -85,B 0,C 180,E1 -17329.518,E2 -17329.518} C_VEL
LIN {X 0,Y 282.074,Z 392.197,A -85,B 0,C 180,E1 -17332.245,E2 -17332.245} C_VEL
LIN {X 0,Y 281.914,Z 394.334,A -85,B 0,C 180,E1 -17333.678,E2 -17333.678} C_VEL
LIN {X 0,Y 283.742,Z 400.399,A -85,B 0,C 180,E1 -17334.157,E2 -17334.157} C_VEL
LIN {X 0,Y 287.649,Z 413.665,A -85,B 0,C 180,E1 -17335.301,E2 -17335.301} C_VEL
LIN {X 0,Y 290.805,Z 427.946,A -85,B 0,C 180,E1 -17336.644,E2 -17336.644} C_VEL
LIN {X 0,Y 292.921,Z 442.283,A -85,B 0,C 180,E1 -17338.14,E2 -17338.14} C_VEL
LIN {X 0,Y 293.842,Z 454.77,A -85,B 0,C 180,E1 -17339.58,E2 -17339.58} C_VEL
LIN {X 0,Y 291.148,Z 468.649,A -85,B 0,C 180,E1 -17341.133,E2 -17341.133} C_VEL
LIN {X 0,Y 288.412,Z 480.859,A -85,B 0,C 180,E1 -17342.812,E2 -17342.812} C_VEL
LIN {X 0,Y 286.002,Z 491.159,A -85,B 0,C 180,E1 -17344.53,E2 -17344.53} C_VEL
LIN {X 0,Y 283.525,Z 501.653,A -85,B 0,C 180,E1 -17346.633,E2 -17346.633} C_VEL
LIN {X 0,Y 281.454,Z 510.534,A -85,B 0,C 180,E1 -17348.772,E2 -17348.772} C_VEL
LIN {X 0,Y 279.261,Z 519.26,A -85,B 0,C 180,E1 -17351.284,E2 -17351.284} C_VEL
LIN {X 0,Y 277.72,Z 526.506,A -85,B 0,C 180,E1 -17353.837,E2 -17353.837} C_VEL
LIN {X 0,Y 276.451,Z 533.204,A -85,B 0,C 180,E1 -17356.773,E2 -17356.773} C_VEL
LIN {X 0,Y 275.682,Z 538.404,A -85,B 0,C 180,E1 -17359.72,E2 -17359.72} C_VEL
LIN {X 0,Y 275.372,Z 542.234,A -85,B 0,C 180,E1 -17362.668,E2 -17362.668} C_VEL
LIN {X 0,Y 275.317,Z 544.762,A -85,B 0,C 180,E1 -17365.608,E2 -17365.608} C_VEL
LIN {X 0,Y 275.366,Z 546.033,A -85,B 0,C 180,E1 -17368.537,E2 -17368.537} C_VEL
LIN {X 0,Y 275.409,Z 546.196,A -85,B 0,C 180,E1 -17370,E2 -17370} C_VEL
LIN {X 0,Y 275.375,Z 545.545,A -85,B 0,C 180,E1 -17372.926,E2 -17372.926} C_VEL
LIN {X 0,Y 275.379,Z 543.637,A -85,B 0,C 180,E1 -17375.859,E2 -17375.859} C_VEL
LIN {X 0,Y 275.491,Z 540.454,A -85,B 0,C 180,E1 -17378.805,E2 -17378.805} C_VEL
LIN {X 0,Y 275.968,Z 535.942,A -85,B 0,C 180,E1 -17381.755,E2 -17381.755} C_VEL
LIN {X 0,Y 276.975,Z 529.994,A -85,B 0,C 180,E1 -17384.699,E2 -17384.699} C_VEL
LIN {X 0,Y 278.558,Z 522.463,A -85,B 0,C 180,E1 -17387.623,E2 -17387.623} C_VEL
LIN {X 0,Y 280.36,Z 514.378,A -85,B 0,C 180,E1 -17390.162,E2 -17390.162} C_VEL
LIN {X 0,Y 282.749,Z 504.655,A -85,B 0,C 180,E1 -17392.66,E2 -17392.66} C_VEL
LIN {X 0,Y 285.082,Z 494.703,A -85,B 0,C 180,E1 -17394.777,E2 -17394.777} C_VEL
LIN {X 0,Y 287.862,Z 482.862,A -85,B 0,C 180,E1 -17396.851,E2 -17396.851} C_VEL
LIN {X 0,Y 290.511,Z 471.049,A -85,B 0,C 180,E1 -17398.541,E2 -17398.541} C_VEL
LIN {X 0,Y 293.21,Z 458.262,A -85,B 0,C 180,E1 -17400.024,E2 -17400.024} C_VEL
LIN {X 0,Y 293.815,Z 453.304,A -85,B 0,C 180,E1 -17400.559,E2 -17400.559} C_VEL
LIN {X 0,Y 292.556,Z 439.542,A -85,B 0,C 180,E1 -17402.135,E2 -17402.135} C_VEL
LIN {X 0,Y 290.229,Z 425.182,A -85,B 0,C 180,E1 -17403.603,E2 -17403.603} C_VEL
LIN {X 0,Y 286.774,Z 410.367,A -85,B 0,C 180,E1 -17404.961,E2 -17404.961} C_VEL
LIN {X 0,Y 282.587,Z 397.049,A -85,B 0,C 180,E1 -17406.091,E2 -17406.091} C_VEL
LIN {X 0,Y 281.853,Z 394.324,A -85,B 0,C 180,E1 -17406.296,E2 -17406.296} C_VEL
LIN {X 0,Y 282.057,Z 392.133,A -85,B 0,C 180,E1 -17407.745,E2 -17407.745} C_VEL
LIN {X 0,Y 281.226,Z 387.036,A -85,B 0,C 180,E1 -17411.434,E2 -17411.434} C_VEL
LIN {X 0,Y 280.317,Z 381.871,A -85,B 0,C 180,E1 -17415.412,E2 -17415.412} C_VEL
LIN {X 0,Y 279.437,Z 377.367,A -85,B 0,C 180,E1 -17419.163,E2 -17419.163} C_VEL
LIN {X 0,Y 278.633,Z 373.398,A -85,B 0,C 180,E1 -17422.746,E2 -17422.746} C_VEL
LIN {X 0,Y 277.853,Z 369.548,A -85,B 0,C 180,E1 -17426.585,E2 -17426.585} C_VEL
LIN {X 0,Y 277.289,Z 366.572,A -85,B 0,C 180,E1 -17429.962,E2 -17429.962} C_VEL
LIN {X 0,Y 277.363,Z 366.562,A -85,B 0,C 180,E1 -17432.865,E2 -17432.865} C_VEL
LIN {X 0,Y 277.331,Z 366.563,A -85,B 0,C 180,E1 -17436.08,E2 -17436.08} C_VEL
LIN {X 0,Y 277.347,Z 366.559,A -85,B 0,C 180,E1 -17440.767,E2 -17440.767} C_VEL
LIN {X 0,Y 277.438,Z 366.551,A -85,B 0,C 180,E1 -17445.326,E2 -17445.326} C_VEL
LIN {X 0,Y 277.463,Z 366.542,A -85,B 0,C 180,E1 -17449.787,E2 -17449.787} C_VEL
LIN {X 0,Y 277.632,Z 366.524,A -85,B 0,C 180,E1 -17452.729,E2 -17452.729} C_VEL
LIN {X 0,Y 277.825,Z 366.504,A -85,B 0,C 180,E1 -17458.551,E2 -17458.551} C_VEL
LIN {X 0,Y 277.824,Z 366.498,A -85,B 0,C 180,E1 -17461.45,E2 -17461.45} C_VEL
LIN {X 0,Y 277.657,Z 366.518,A -85,B 0,C 180,E1 -17467.271,E2 -17467.271} C_VEL
LIN {X 0,Y 277.511,Z 366.541,A -85,B 0,C 180,E1 -17470.211,E2 -17470.211} C_VEL
LIN {X 0,Y 277.439,Z 366.545,A -85,B 0,C 180,E1 -17474.674,E2 -17474.674} C_VEL
LIN {X 0,Y 277.348,Z 366.562,A -85,B 0,C 180,E1 -17479.234,E2 -17479.234} C_VEL
LIN {X 0,Y 277.322,Z 366.559,A -85,B 0,C 180,E1 -17484.171,E2 -17484.171} C_VEL
LIN {X 0,Y 277.329,Z 366.561,A -85,B 0,C 180,E1 -17487.506,E2 -17487.506} C_VEL
LIN {X 0,Y 277.274,Z 366.57,A -85,B 0,C 180,E1 -17490.481,E2 -17490.481} C_VEL
LIN {X 0,Y 277.25,Z 366.575,A -85,B 0,C 180,E1 -17493.896,E2 -17493.896} C_VEL
LIN {X 0,Y 277.325,Z 366.651,A -85,B 0,C 180,E1 -17496.56,E2 -17496.56} C_VEL
LIN {X 0,Y 277.871,Z 370.069,A -85,B 0,C 180,E1 -17501.118,E2 -17501.118} C_VEL
LIN {X 0,Y 278.387,Z 373.267,A -85,B 0,C 180,E1 -17505.019,E2 -17505.019} C_VEL
LIN {X 0,Y 278.62,Z 375.062,A -85,B 0,C 180,E1 -17507.074,E2 -17507.074} C_VEL
LIN {X 0,Y 278.796,Z 376.941,A -85,B 0,C 180,E1 -17509.135,E2 -17509.135} C_VEL
LIN {X 0,Y 278.778,Z 379.123,A -85,B 0,C 180,E1 -17511.4,E2 -17511.4} C_VEL
LIN {X 0,Y 278.477,Z 382.342,A -85,B 0,C 180,E1 -17514.517,E2 -17514.517} C_VEL
LIN {X 0,Y 278.301,Z 383.848,A -85,B 0,C 180,E1 -17515.92,E2 -17515.92} C_VEL
LIN {X 0,Y 279.501,Z 387.217,A -85,B 0,C 180,E1 -17516.238,E2 -17516.238} C_VEL
LIN {X 0,Y 284.333,Z 398.653,A -85,B 0,C 180,E1 -17517.423,E2 -17517.423} C_VEL
LIN {X 0,Y 288.709,Z 411.463,A -85,B 0,C 180,E1 -17518.81,E2 -17518.81} C_VEL
LIN {X 0,Y 292.119,Z 424.597,A -85,B 0,C 180,E1 -17520.337,E2 -17520.337} C_VEL
LIN {X 0,Y 294.445,Z 437.834,A -85,B 0,C 180,E1 -17522.024,E2 -17522.024} C_VEL
LIN {X 0,Y 293.63,Z 443.837,A -85,B 0,C 180,E1 -17522.684,E2 -17522.684} C_VEL
LIN {X 0,Y 291.227,Z 456.31,A -85,B 0,C 180,E1 -17524.254,E2 -17524.254} C_VEL
LIN {X 0,Y 288.651,Z 467.221,A -85,B 0,C 180,E1 -17525.932,E2 -17525.932} C_VEL
LIN {X 0,Y 286.031,Z 477.993,A -85,B 0,C 180,E1 -17527.994,E2 -17527.994} C_VEL
LIN {X 0,Y 283.546,Z 487.293,A -85,B 0,C 180,E1 -17530.182,E2 -17530.182} C_VEL
LIN {X 0,Y 281.435,Z 495.446,A -85,B 0,C 180,E1 -17532.563,E2 -17532.563} C_VEL
LIN {X 0,Y 279.708,Z 501.495,A -85,B 0,C 180,E1 -17534.703,E2 -17534.703} C_VEL
LIN {X 0,Y 277.988,Z 507.929,A -85,B 0,C 180,E1 -17537.591,E2 -17537.591} C_VEL
LIN {X 0,Y 276.807,Z 512.786,A -85,B 0,C 180,E1 -17540.501,E2 -17540.501} C_VEL
LIN {X 0,Y 276.204,Z 515.744,A -85,B 0,C 180,E1 -17542.912,E2 -17542.912} C_VEL
LIN {X 0,Y 275.748,Z 517.99,A -85,B 0,C 180,E1 -17545.615,E2 -17545.615} C_VEL
LIN {X 0,Y 275.475,Z 519.216,A -85,B 0,C 180,E1 -17548.538,E2 -17548.538} C_VEL
LIN {X 0,Y 275.474,Z 519.238,A -85,B 0,C 180,E1 -17551.462,E2 -17551.462} C_VEL
LIN {X 0,Y 275.743,Z 518.061,A -85,B 0,C 180,E1 -17554.385,E2 -17554.385} C_VEL
LIN {X 0,Y 276.221,Z 515.649,A -85,B 0,C 180,E1 -17557.309,E2 -17557.309} C_VEL
LIN {X 0,Y 277.042,Z 511.917,A -85,B 0,C 180,E1 -17560.229,E2 -17560.229} C_VEL
LIN {X 0,Y 278.34,Z 506.731,A -85,B 0,C 180,E1 -17563.135,E2 -17563.135} C_VEL
LIN {X 0,Y 279.667,Z 501.777,A -85,B 0,C 180,E1 -17565.3,E2 -17565.3} C_VEL
LIN {X 0,Y 281.731,Z 494.698,A -85,B 0,C 180,E1 -17567.794,E2 -17567.794} C_VEL
LIN {X 0,Y 283.554,Z 487.315,A -85,B 0,C 180,E1 -17569.93,E2 -17569.93} C_VEL
LIN {X 0,Y 285.954,Z 478.493,A -85,B 0,C 180,E1 -17572.013,E2 -17572.013} C_VEL
LIN {X 0,Y 288.552,Z 467.819,A -85,B 0,C 180,E1 -17574.077,E2 -17574.077} C_VEL
LIN {X 0,Y 291.084,Z 457.029,A -85,B 0,C 180,E1 -17575.76,E2 -17575.76} C_VEL
LIN {X 0,Y 293.557,Z 444.876,A -85,B 0,C 180,E1 -17577.302,E2 -17577.302} C_VEL
LIN {X 0,Y 294.551,Z 438.401,A -85,B 0,C 180,E1 -17578.015,E2 -17578.015} C_VEL
LIN {X 0,Y 292.557,Z 426.552,A -85,B 0,C 180,E1 -17579.537,E2 -17579.537} C_VEL
LIN {X 0,Y 289.244,Z 413.16,A -85,B 0,C 180,E1 -17581.112,E2 -17581.112} C_VEL
LIN {X 0,Y 284.725,Z 399.664,A -85,B 0,C 180,E1 -17582.591,E2 -17582.591} C_VEL
LIN {X 0,Y 279.586,Z 387.273,A -85,B 0,C 180,E1 -17583.876,E2 -17583.876} C_VEL
LIN {X 0,Y 278.44,Z 384.587,A -85,B 0,C 180,E1 -17584.139,E2 -17584.139} C_VEL
LIN {X 0,Y 278.323,Z 383.814,A -85,B 0,C 180,E1 -17584.233,E2 -17584.233} C_VEL
LIN {X 0,Y 278.668,Z 380.623,A -85,B 0,C 180,E1 -17587.25,E2 -17587.25} C_VEL
LIN {X 0,Y 278.79,Z 378.816,A -85,B 0,C 180,E1 -17589.067,E2 -17589.067} C_VEL
LIN {X 0,Y 278.785,Z 377.02,A -85,B 0,C 180,E1 -17590.954,E2 -17590.954} C_VEL
LIN {X 0,Y 278.612,Z 375.183,A -85,B 0,C 180,E1 -17592.985,E2 -17592.985} C_VEL
LIN {X 0,Y 278.123,Z 371.734,A -85,B 0,C 180,E1 -17596.978,E2 -17596.978} C_VEL
LIN {X 0,Y 277.65,Z 368.75,A -85,B 0,C 180,E1 -17600.742,E2 -17600.742} C_VEL
LIN {X 0,Y 277.288,Z 366.57,A -85,B 0,C 180,E1 -17603.88,E2 -17603.88} C_VEL
LIN {X 0,Y 277.249,Z 366.573,A -85,B 0,C 180,E1 -17607.837,E2 -17607.837} C_VEL
LIN {X 0,Y 277.294,Z 366.568,A -85,B 0,C 180,E1 -17611.213,E2 -17611.213} C_VEL
LIN {X 0,Y 277.318,Z 366.563,A -85,B 0,C 180,E1 -17614.48,E2 -17614.48} C_VEL
LIN {X 0,Y 277.29,Z 366.571,A -85,B 0,C 180,E1 -17617.655,E2 -17617.655} C_VEL
LIN {X 0,Y 277.349,Z 366.563,A -85,B 0,C 180,E1 -17620.766,E2 -17620.766} C_VEL
LIN {X 0,Y 277.439,Z 366.546,A -85,B 0,C 180,E1 -17625.326,E2 -17625.326} C_VEL
LIN {X 0,Y 277.511,Z 366.543,A -85,B 0,C 180,E1 -17629.789,E2 -17629.789} C_VEL
LIN {X 0,Y 277.658,Z 366.524,A -85,B 0,C 180,E1 -17632.729,E2 -17632.729} C_VEL
LIN {X 0,Y 277.825,Z 366.497,A -85,B 0,C 180,E1 -17638.55,E2 -17638.55} C_VEL
LIN {X 0,Y 277.825,Z 366.497,A -85,B 0,C 180,E1 -17641.449,E2 -17641.449} C_VEL
LIN {X 0,Y 277.682,Z 366.52,A -85,B 0,C 180,E1 -17642.994,E2 -17642.994} C_VEL
LIN {X 0,Y 276.859,Z 366.619,A -85,B 0,C 180,E1 -17644.203,E2 -17644.203} C_VEL
LIN {X 0,Y 274.02,Z 366.978,A -85,B 0,C 180,E1 -17646.176,E2 -17646.176} C_VEL
LIN {X 0,Y 270.865,Z 367.375,A -85,B 0,C 180,E1 -17648.601,E2 -17648.601} C_VEL
LIN {X 0,Y 270.494,Z 367.416,A -85,B 0,C 180,E1 -17649.438,E2 -17649.438} C_VEL
LIN {X 0,Y 270.365,Z 367.433,A -85,B 0,C 180,E1 -17653.53,E2 -17653.53} C_VEL
LIN {X 0,Y 270.359,Z 367.434,A -85,B 0,C 180,E1 -17656.615,E2 -17656.615} C_VEL
LIN {X 0,Y 270.303,Z 367.442,A -85,B 0,C 180,E1 -17660.605,E2 -17660.605} C_VEL
LIN {X 0,Y 270.277,Z 367.443,A -85,B 0,C 180,E1 -17664.585,E2 -17664.585} C_VEL
LIN {X 0,Y 270.254,Z 367.498,A -85,B 0,C 180,E1 -17668.757,E2 -17668.757} C_VEL
LIN {X 0,Y 270.952,Z 371.176,A -85,B 0,C 180,E1 -17673.004,E2 -17673.004} C_VEL
LIN {X 0,Y 271.675,Z 374.719,A -85,B 0,C 180,E1 -17676.683,E2 -17676.683} C_VEL
LIN {X 0,Y 272.414,Z 378.422,A -85,B 0,C 180,E1 -17680.163,E2 -17680.163} C_VEL
LIN {X 0,Y 273.268,Z 382.835,A -85,B 0,C 180,E1 -17683.979,E2 -17683.979} C_VEL
LIN {X 0,Y 274.212,Z 388.122,A -85,B 0,C 180,E1 -17688.212,E2 -17688.212} C_VEL
LIN {X 0,Y 274.926,Z 392.131,A -85,B 0,C 180,E1 -17691.222,E2 -17691.222} C_VEL
LIN {X 0,Y 275.114,Z 394.216,A -85,B 0,C 180,E1 -17692.695,E2 -17692.695} C_VEL
LIN {X 0,Y 276.318,Z 397.641,A -85,B 0,C 180,E1 -17692.994,E2 -17692.994} C_VEL
LIN {X 0,Y 280.758,Z 412.143,A -85,B 0,C 180,E1 -17694.29,E2 -17694.29} C_VEL
LIN {X 0,Y 283.968,Z 426.291,A -85,B 0,C 180,E1 -17695.658,E2 -17695.658} C_VEL
LIN {X 0,Y 286.139,Z 439.809,A -85,B 0,C 180,E1 -17697.107,E2 -17697.107} C_VEL
LIN {X 0,Y 287.257,Z 452.558,A -85,B 0,C 180,E1 -17698.613,E2 -17698.613} C_VEL
LIN {X 0,Y 287.309,Z 456.425,A -85,B 0,C 180,E1 -17699.09,E2 -17699.09} C_VEL
LIN {X 0,Y 284.604,Z 469.493,A -85,B 0,C 180,E1 -17700.607,E2 -17700.607} C_VEL
LIN {X 0,Y 281.786,Z 481.516,A -85,B 0,C 180,E1 -17702.32,E2 -17702.32} C_VEL
LIN {X 0,Y 279.057,Z 492.632,A -85,B 0,C 180,E1 -17704.25,E2 -17704.25} C_VEL
LIN {X 0,Y 276.42,Z 503.393,A -85,B 0,C 180,E1 -17706.531,E2 -17706.531} C_VEL
LIN {X 0,Y 274.033,Z 512.843,A -85,B 0,C 180,E1 -17708.958,E2 -17708.958} C_VEL
LIN {X 0,Y 271.954,Z 521.141,A -85,B 0,C 180,E1 -17711.544,E2 -17711.544} C_VEL
LIN {X 0,Y 270.321,Z 528.386,A -85,B 0,C 180,E1 -17714.324,E2 -17714.324} C_VEL
LIN {X 0,Y 269.214,Z 534.323,A -85,B 0,C 180,E1 -17717.179,E2 -17717.179} C_VEL
LIN {X 0,Y 268.515,Z 539.167,A -85,B 0,C 180,E1 -17720.204,E2 -17720.204} C_VEL
LIN {X 0,Y 268.29,Z 541.886,A -85,B 0,C 180,E1 -17722.474,E2 -17722.474} C_VEL
LIN {X 0,Y 268.228,Z 544.416,A -85,B 0,C 180,E1 -17725.491,E2 -17725.491} C_VEL
LIN {X 0,Y 268.288,Z 545.688,A -85,B 0,C 180,E1 -17728.499,E2 -17728.499} C_VEL
LIN {X 0,Y 268.327,Z 545.851,A -85,B 0,C 180,E1 -17730,E2 -17730} C_VEL
LIN {X 0,Y 268.28,Z 545.199,A -85,B 0,C 180,E1 -17733.003,E2 -17733.003} C_VEL
LIN {X 0,Y 268.291,Z 543.289,A -85,B 0,C 180,E1 -17736.014,E2 -17736.014} C_VEL
LIN {X 0,Y 268.423,Z 540.104,A -85,B 0,C 180,E1 -17739.038,E2 -17739.038} C_VEL
LIN {X 0,Y 268.967,Z 535.588,A -85,B 0,C 180,E1 -17742.066,E2 -17742.066} C_VEL
LIN {X 0,Y 270.016,Z 529.635,A -85,B 0,C 180,E1 -17745.087,E2 -17745.087} C_VEL
LIN {X 0,Y 271.715,Z 522.098,A -85,B 0,C 180,E1 -17748.082,E2 -17748.082} C_VEL
LIN {X 0,Y 273.651,Z 514.006,A -85,B 0,C 180,E1 -17750.679,E2 -17750.679} C_VEL
LIN {X 0,Y 276.093,Z 504.432,A -85,B 0,C 180,E1 -17753.196,E2 -17753.196} C_VEL
LIN {X 0,Y 278.583,Z 494.302,A -85,B 0,C 180,E1 -17755.396,E2 -17755.396} C_VEL
LIN {X 0,Y 281.512,Z 482.439,A -85,B 0,C 180,E1 -17757.507,E2 -17757.507} C_VEL
LIN {X 0,Y 284.258,Z 470.595,A -85,B 0,C 180,E1 -17759.229,E2 -17759.229} C_VEL
LIN {X 0,Y 287.245,Z 456.74,A -85,B 0,C 180,E1 -17760.846,E2 -17760.846} C_VEL
LIN {X 0,Y 287.03,Z 449.577,A -85,B 0,C 180,E1 -17761.724,E2 -17761.724} C_VEL
LIN {X 0,Y 285.645,Z 436.53,A -85,B 0,C 180,E1 -17763.224,E2 -17763.224} C_VEL
LIN {X 0,Y 283.106,Z 422.186,A -85,B 0,C 180,E1 -17764.715,E2 -17764.715} C_VEL
LIN {X 0,Y 279.63,Z 408.278,A -85,B 0,C 180,E1 -17766.032,E2 -17766.032} C_VEL
LIN {X 0,Y 275.908,Z 396.977,A -85,B 0,C 180,E1 -17767.053,E2 -17767.053} C_VEL
LIN {X 0,Y 275.076,Z 394.065,A -85,B 0,C 180,E1 -17767.322,E2 -17767.322} C_VEL
LIN {X 0,Y 274.647,Z 390.611,A -85,B 0,C 180,E1 -17769.855,E2 -17769.855} C_VEL
LIN {X 0,Y 273.706,Z 385.191,A -85,B 0,C 180,E1 -17774.032,E2 -17774.032} C_VEL
LIN {X 0,Y 272.807,Z 380.485,A -85,B 0,C 180,E1 -17777.948,E2 -17777.948} C_VEL
LIN {X 0,Y 271.998,Z 376.36,A -85,B 0,C 180,E1 -17781.675,E2 -17781.675} C_VEL
LIN {X 0,Y 271.282,Z 372.718,A -85,B 0,C 180,E1 -17785.254,E2 -17785.254} C_VEL
LIN {X 0,Y 270.577,Z 369.311,A -85,B 0,C 180,E1 -17788.998,E2 -17788.998} C_VEL
LIN {X 0,Y 270.251,Z 367.452,A -85,B 0,C 180,E1 -17791.243,E2 -17791.243} C_VEL
LIN {X 0,Y 270.279,Z 367.445,A -85,B 0,C 180,E1 -17795.519,E2 -17795.519} C_VEL
LIN {X 0,Y 270.304,Z 367.44,A -85,B 0,C 180,E1 -17800.245,E2 -17800.245} C_VEL
LIN {X 0,Y 270.406,Z 367.423,A -85,B 0,C 180,E1 -17804.936,E2 -17804.936} C_VEL
LIN {X 0,Y 270.415,Z 367.422,A -85,B 0,C 180,E1 -17809.518,E2 -17809.518} C_VEL
LIN {X 0,Y 270.589,Z 367.403,A -85,B 0,C 180,E1 -17812.538,E2 -17812.538} C_VEL
LIN {X 0,Y 270.79,Z 367.38,A -85,B 0,C 180,E1 -17818.513,E2 -17818.513} C_VEL
LIN {X 0,Y 270.79,Z 367.374,A -85,B 0,C 180,E1 -17821.487,E2 -17821.487} C_VEL
LIN {X 0,Y 270.615,Z 367.394,A -85,B 0,C 180,E1 -17827.461,E2 -17827.461} C_VEL
LIN {X 0,Y 270.446,Z 367.419,A -85,B 0,C 180,E1 -17830.481,E2 -17830.481} C_VEL
LIN {X 0,Y 270.406,Z 367.42,A -85,B 0,C 180,E1 -17835.065,E2 -17835.065} C_VEL
LIN {X 0,Y 270.305,Z 367.441,A -85,B 0,C 180,E1 -17839.756,E2 -17839.756} C_VEL
LIN {X 0,Y 270.277,Z 367.437,A -85,B 0,C 180,E1 -17844.586,E2 -17844.586} C_VEL
LIN {X 0,Y 270.275,Z 367.442,A -85,B 0,C 180,E1 -17847.909,E2 -17847.909} C_VEL
LIN {X 0,Y 270.187,Z 367.454,A -85,B 0,C 180,E1 -17851.348,E2 -17851.348} C_VEL
LIN {X 0,Y 270.234,Z 367.54,A -85,B 0,C 180,E1 -17855.438,E2 -17855.438} C_VEL
LIN {X 0,Y 270.656,Z 369.928,A -85,B 0,C 180,E1 -17858.831,E2 -17858.831} C_VEL
LIN {X 0,Y 271.087,Z 372.625,A -85,B 0,C 180,E1 -17862.381,E2 -17862.381} C_VEL
LIN {X 0,Y 271.588,Z 375.959,A -85,B 0,C 180,E1 -17866.433,E2 -17866.433} C_VEL
LIN {X 0,Y 271.814,Z 378.903,A -85,B 0,C 180,E1 -17869.729,E2 -17869.729} C_VEL
LIN {X 0,Y 271.627,Z 382.423,A -85,B 0,C 180,E1 -17873.33,E2 -17873.33} C_VEL
LIN {X 0,Y 271.441,Z 384.178,A -85,B 0,C 180,E1 -17874.912,E2 -17874.912} C_VEL
LIN {X 0,Y 272.622,Z 387.387,A -85,B 0,C 180,E1 -17875.214,E2 -17875.214} C_VEL
LIN {X 0,Y 277.722,Z 399.211,A -85,B 0,C 180,E1 -17876.521,E2 -17876.521} C_VEL
LIN {X 0,Y 281.993,Z 411.578,A -85,B 0,C 180,E1 -17877.927,E2 -17877.927} C_VEL
LIN {X 0,Y 285.036,Z 422.891,A -85,B 0,C 180,E1 -17879.296,E2 -17879.296} C_VEL
LIN {X 0,Y 287.419,Z 435.071,A -85,B 0,C 180,E1 -17880.88,E2 -17880.88} C_VEL
LIN {X 0,Y 288.106,Z 440.166,A -85,B 0,C 180,E1 -17881.584,E2 -17881.584} C_VEL
LIN {X 0,Y 285.645,Z 453.036,A -85,B 0,C 180,E1 -17883.122,E2 -17883.122} C_VEL
LIN {X 0,Y 283.217,Z 463.505,A -85,B 0,C 180,E1 -17884.656,E2 -17884.656} C_VEL
LIN {X 0,Y 280.827,Z 473.264,A -85,B 0,C 180,E1 -17886.396,E2 -17886.396} C_VEL
LIN {X 0,Y 278.173,Z 483.036,A -85,B 0,C 180,E1 -17888.51,E2 -17888.51} C_VEL
LIN {X 0,Y 275.569,Z 492.373,A -85,B 0,C 180,E1 -17891.024,E2 -17891.024} C_VEL
LIN {X 0,Y 273.441,Z 499.946,A -85,B 0,C 180,E1 -17893.577,E2 -17893.577} C_VEL
LIN {X 0,Y 271.92,Z 505.273,A -85,B 0,C 180,E1 -17895.787,E2 -17895.787} C_VEL
LIN {X 0,Y 270.378,Z 510.893,A -85,B 0,C 180,E1 -17898.758,E2 -17898.758} C_VEL
LIN {X 0,Y 269.578,Z 514.155,A -85,B 0,C 180,E1 -17901.001,E2 -17901.001} C_VEL
LIN {X 0,Y 268.917,Z 517.262,A -85,B 0,C 180,E1 -17904,E2 -17904} C_VEL
LIN {X 0,Y 268.499,Z 519.1,A -85,B 0,C 180,E1 -17906.999,E2 -17906.999} C_VEL
LIN {X 0,Y 268.343,Z 519.722,A -85,B 0,C 180,E1 -17910,E2 -17910} C_VEL
LIN {X 0,Y 268.498,Z 519.146,A -85,B 0,C 180,E1 -17913.001,E2 -17913.001} C_VEL
LIN {X 0,Y 268.9,Z 517.359,A -85,B 0,C 180,E1 -17916.001,E2 -17916.001} C_VEL
LIN {X 0,Y 269.575,Z 514.3,A -85,B 0,C 180,E1 -17919,E2 -17919} C_VEL
LIN {X 0,Y 270.692,Z 509.866,A -85,B 0,C 180,E1 -17921.988,E2 -17921.988} C_VEL
LIN {X 0,Y 272.273,Z 503.892,A -85,B 0,C 180,E1 -17924.959,E2 -17924.959} C_VEL
LIN {X 0,Y 274.337,Z 497.243,A -85,B 0,C 180,E1 -17927.519,E2 -17927.519} C_VEL
LIN {X 0,Y 276.457,Z 489.293,A -85,B 0,C 180,E1 -17929.994,E2 -17929.994} C_VEL
LIN {X 0,Y 278.915,Z 480.486,A -85,B 0,C 180,E1 -17932.208,E2 -17932.208} C_VEL
LIN {X 0,Y 281.631,Z 470.157,A -85,B 0,C 180,E1 -17934.315,E2 -17934.315} C_VEL
LIN {X 0,Y 284.248,Z 459.794,A -85,B 0,C 180,E1 -17936.032,E2 -17936.032} C_VEL
LIN {X 0,Y 286.613,Z 448.587,A -85,B 0,C 180,E1 -17937.57,E2 -17937.57} C_VEL
LIN {X 0,Y 288.123,Z 439.812,A -85,B 0,C 180,E1 -17938.582,E2 -17938.582} C_VEL
LIN {X 0,Y 286.221,Z 428.164,A -85,B 0,C 180,E1 -17940.152,E2 -17940.152} C_VEL
LIN {X 0,Y 283.191,Z 415.482,A -85,B 0,C 180,E1 -17941.722,E2 -17941.722} C_VEL
LIN {X 0,Y 279.04,Z 402.739,A -85,B 0,C 180,E1 -17943.21,E2 -17943.21} C_VEL
LIN {X 0,Y 274.358,Z 391.046,A -85,B 0,C 180,E1 -17944.515,E2 -17944.515} C_VEL
LIN {X 0,Y 272.578,Z 387.252,A -85,B 0,C 180,E1 -17944.93,E2 -17944.93} C_VEL
LIN {X 0,Y 271.467,Z 384.017,A -85,B 0,C 180,E1 -17945.25,E2 -17945.25} C_VEL
LIN {X 0,Y 271.834,Z 380.109,A -85,B 0,C 180,E1 -17949.138,E2 -17949.138} C_VEL
LIN {X 0,Y 271.709,Z 377.28,A -85,B 0,C 180,E1 -17952.262,E2 -17952.262} C_VEL
LIN {X 0,Y 271.354,Z 374.372,A -85,B 0,C 180,E1 -17955.629,E2 -17955.629} C_VEL
LIN {X 0,Y 270.878,Z 371.244,A -85,B 0,C 180,E1 -17959.561,E2 -17959.561} C_VEL
LIN {X 0,Y 270.439,Z 368.524,A -85,B 0,C 180,E1 -17963.294,E2 -17963.294} C_VEL
LIN {X 0,Y 270.206,Z 367.454,A -85,B 0,C 180,E1 -17965.095,E2 -17965.095} C_VEL
LIN {X 0,Y 270.204,Z 367.451,A -85,B 0,C 180,E1 -17969.131,E2 -17969.131} C_VEL
LIN {X 0,Y 270.269,Z 367.443,A -85,B 0,C 180,E1 -17972.146,E2 -17972.146} C_VEL
LIN {X 0,Y 270.281,Z 367.443,A -85,B 0,C 180,E1 -17975.519,E2 -17975.519} C_VEL
LIN {X 0,Y 270.306,Z 367.44,A -85,B 0,C 180,E1 -17980.244,E2 -17980.244} C_VEL
LIN {X 0,Y 270.408,Z 367.421,A -85,B 0,C 180,E1 -17984.935,E2 -17984.935} C_VEL
LIN {X 0,Y 270.446,Z 367.422,A -85,B 0,C 180,E1 -17989.519,E2 -17989.519} C_VEL
LIN {X 0,Y 270.616,Z 367.4,A -85,B 0,C 180,E1 -17992.539,E2 -17992.539} C_VEL
LIN {X 0,Y 270.791,Z 367.373,A -85,B 0,C 180,E1 -17998.513,E2 -17998.513} C_VEL
LIN {X 0,Y 270.791,Z 367.373,A -85,B 0,C 180,E1 -18001.487,E2 -18001.487} C_VEL
LIN {X 0,Y 270.589,Z 367.4,A -85,B 0,C 180,E1 -18007.462,E2 -18007.462} C_VEL
LIN {X 0,Y 270.494,Z 367.416,A -85,B 0,C 180,E1 -18009.438,E2 -18009.438} C_VEL
LIN {X 0,Y 269.726,Z 367.51,A -85,B 0,C 180,E1 -18010.679,E2 -18010.679} C_VEL
LIN {X 0,Y 266.824,Z 367.879,A -85,B 0,C 180,E1 -18012.702,E2 -18012.702} C_VEL
LIN {X 0,Y 264.43,Z 368.179,A -85,B 0,C 180,E1 -18014.346,E2 -18014.346} C_VEL
LIN {X 0,Y 263.424,Z 368.304,A -85,B 0,C 180,E1 -18015.621,E2 -18015.621} C_VEL
LIN {X 0,Y 263.35,Z 368.311,A -85,B 0,C 180,E1 -18016.053,E2 -18016.053} C_VEL
LIN {X 0,Y 263.255,Z 368.323,A -85,B 0,C 180,E1 -18020.87,E2 -18020.87} C_VEL
LIN {X 0,Y 263.212,Z 368.32,A -85,B 0,C 180,E1 -18025.291,E2 -18025.291} C_VEL
LIN {X 0,Y 263.22,Z 368.411,A -85,B 0,C 180,E1 -18027.322,E2 -18027.322} C_VEL
LIN {X 0,Y 263.827,Z 371.764,A -85,B 0,C 180,E1 -18031.521,E2 -18031.521} C_VEL
LIN {X 0,Y 264.409,Z 374.474,A -85,B 0,C 180,E1 -18034.514,E2 -18034.514} C_VEL
LIN {X 0,Y 264.995,Z 377.464,A -85,B 0,C 180,E1 -18037.588,E2 -18037.588} C_VEL
LIN {X 0,Y 265.791,Z 381.483,A -85,B 0,C 180,E1 -18041.379,E2 -18041.379} C_VEL
LIN {X 0,Y 266.648,Z 386.107,A -85,B 0,C 180,E1 -18045.368,E2 -18045.368} C_VEL
LIN {X 0,Y 267.415,Z 390.506,A -85,B 0,C 180,E1 -18048.925,E2 -18048.925} C_VEL
LIN {X 0,Y 268.042,Z 394.038,A -85,B 0,C 180,E1 -18051.59,E2 -18051.59} C_VEL
LIN {X 0,Y 269.237,Z 397.228,A -85,B 0,C 180,E1 -18051.896,E2 -18051.896} C_VEL
LIN {X 0,Y 270.642,Z 400.347,A -85,B 0,C 180,E1 -18052.24,E2 -18052.24} C_VEL
LIN {X 0,Y 274.737,Z 413.68,A -85,B 0,C 180,E1 -18053.533,E2 -18053.533} C_VEL
LIN {X 0,Y 277.713,Z 427.302,A -85,B 0,C 180,E1 -18054.917,E2 -18054.917} C_VEL
LIN {X 0,Y 279.829,Z 441.071,A -85,B 0,C 180,E1 -18056.458,E2 -18056.458} C_VEL
LIN {X 0,Y 280.856,Z 453.621,A -85,B 0,C 180,E1 -18058.004,E2 -18058.004} C_VEL
LIN {X 0,Y 280.817,Z 457.779,A -85,B 0,C 180,E1 -18058.539,E2 -18058.539} C_VEL
LIN {X 0,Y 278.095,Z 470.338,A -85,B 0,C 180,E1 -18060.058,E2 -18060.058} C_VEL
LIN {X 0,Y 274.905,Z 483.25,A -85,B 0,C 180,E1 -18061.981,E2 -18061.981} C_VEL
LIN {X 0,Y 272.119,Z 494.038,A -85,B 0,C 180,E1 -18063.956,E2 -18063.956} C_VEL
LIN {X 0,Y 269.448,Z 504.47,A -85,B 0,C 180,E1 -18066.28,E2 -18066.28} C_VEL
LIN {X 0,Y 266.965,Z 513.73,A -85,B 0,C 180,E1 -18068.778,E2 -18068.778} C_VEL
LIN {X 0,Y 264.868,Z 521.814,A -85,B 0,C 180,E1 -18071.433,E2 -18071.433} C_VEL
LIN {X 0,Y 263.125,Z 529.339,A -85,B 0,C 180,E1 -18074.508,E2 -18074.508} C_VEL
LIN {X 0,Y 261.972,Z 535.277,A -85,B 0,C 180,E1 -18077.607,E2 -18077.607} C_VEL
LIN {X 0,Y 261.374,Z 539.788,A -85,B 0,C 180,E1 -18080.716,E2 -18080.716} C_VEL
LIN {X 0,Y 261.15,Z 542.964,A -85,B 0,C 180,E1 -18083.82,E2 -18083.82} C_VEL
LIN {X 0,Y 261.184,Z 544.864,A -85,B 0,C 180,E1 -18086.915,E2 -18086.915} C_VEL
LIN {X 0,Y 261.247,Z 545.507,A -85,B 0,C 180,E1 -18090,E2 -18090} C_VEL
LIN {X 0,Y 261.187,Z 544.853,A -85,B 0,C 180,E1 -18093.085,E2 -18093.085} C_VEL
LIN {X 0,Y 261.212,Z 542.941,A -85,B 0,C 180,E1 -18096.178,E2 -18096.178} C_VEL
LIN {X 0,Y 261.374,Z 539.754,A -85,B 0,C 180,E1 -18099.284,E2 -18099.284} C_VEL
LIN {X 0,Y 261.97,Z 535.235,A -85,B 0,C 180,E1 -18102.393,E2 -18102.393} C_VEL
LIN {X 0,Y 263.074,Z 529.276,A -85,B 0,C 180,E1 -18105.495,E2 -18105.495} C_VEL
LIN {X 0,Y 264.866,Z 521.732,A -85,B 0,C 180,E1 -18108.567,E2 -18108.567} C_VEL
LIN {X 0,Y 266.945,Z 513.634,A -85,B 0,C 180,E1 -18111.223,E2 -18111.223} C_VEL
LIN {X 0,Y 269.398,Z 504.423,A -85,B 0,C 180,E1 -18113.706,E2 -18113.706} C_VEL
LIN {X 0,Y 272.086,Z 493.899,A -85,B 0,C 180,E1 -18116.047,E2 -18116.047} C_VEL
LIN {X 0,Y 275.178,Z 482.016,A -85,B 0,C 180,E1 -18118.196,E2 -18118.196} C_VEL
LIN {X 0,Y 278.046,Z 470.14,A -85,B 0,C 180,E1 -18119.948,E2 -18119.948} C_VEL
LIN {X 0,Y 280.814,Z 457.723,A -85,B 0,C 180,E1 -18121.435,E2 -18121.435} C_VEL
LIN {X 0,Y 280.35,Z 446.572,A -85,B 0,C 180,E1 -18122.852,E2 -18122.852} C_VEL
LIN {X 0,Y 278.768,Z 433.511,A -85,B 0,C 180,E1 -18124.377,E2 -18124.377} C_VEL
LIN {X 0,Y 275.891,Z 418.536,A -85,B 0,C 180,E1 -18125.959,E2 -18125.959} C_VEL
LIN {X 0,Y 271.78,Z 403.68,A -85,B 0,C 180,E1 -18127.408,E2 -18127.408} C_VEL
LIN {X 0,Y 269.483,Z 397.614,A -85,B 0,C 180,E1 -18128.008,E2 -18128.008} C_VEL
LIN {X 0,Y 268.079,Z 394.332,A -85,B 0,C 180,E1 -18128.351,E2 -18128.351} C_VEL
LIN {X 0,Y 268,Z 393.925,A -85,B 0,C 180,E1 -18128.399,E2 -18128.399} C_VEL
LIN {X 0,Y 267.115,Z 388.593,A -85,B 0,C 180,E1 -18132.549,E2 -18132.549} C_VEL
LIN {X 0,Y 266.212,Z 383.651,A -85,B 0,C 180,E1 -18136.655,E2 -18136.655} C_VEL
LIN {X 0,Y 265.385,Z 379.324,A -85,B 0,C 180,E1 -18140.538,E2 -18140.538} C_VEL
LIN {X 0,Y 264.614,Z 375.57,A -85,B 0,C 180,E1 -18144.246,E2 -18144.246} C_VEL
LIN {X 0,Y 263.935,Z 372.289,A -85,B 0,C 180,E1 -18147.822,E2 -18147.822} C_VEL
LIN {X 0,Y 263.267,Z 368.569,A -85,B 0,C 180,E1 -18152.365,E2 -18152.365} C_VEL
LIN {X 0,Y 263.196,Z 368.327,A -85,B 0,C 180,E1 -18153.003,E2 -18153.003} C_VEL
LIN {X 0,Y 263.186,Z 368.323,A -85,B 0,C 180,E1 -18156.387,E2 -18156.387} C_VEL
LIN {X 0,Y 263.266,Z 368.314,A -85,B 0,C 180,E1 -18159.694,E2 -18159.694} C_VEL
LIN {X 0,Y 263.353,Z 368.298,A -85,B 0,C 180,E1 -18164.522,E2 -18164.522} C_VEL
LIN {X 0,Y 263.358,Z 368.303,A -85,B 0,C 180,E1 -18169.234,E2 -18169.234} C_VEL
LIN {X 0,Y 263.548,Z 368.282,A -85,B 0,C 180,E1 -18172.338,E2 -18172.338} C_VEL
LIN {X 0,Y 263.755,Z 368.256,A -85,B 0,C 180,E1 -18178.473,E2 -18178.473} C_VEL
LIN {X 0,Y 263.754,Z 368.25,A -85,B 0,C 180,E1 -18181.527,E2 -18181.527} C_VEL
LIN {X 0,Y 263.576,Z 368.27,A -85,B 0,C 180,E1 -18187.662,E2 -18187.662} C_VEL
LIN {X 0,Y 263.378,Z 368.297,A -85,B 0,C 180,E1 -18190.766,E2 -18190.766} C_VEL
LIN {X 0,Y 263.354,Z 368.3,A -85,B 0,C 180,E1 -18195.478,E2 -18195.478} C_VEL
LIN {X 0,Y 263.267,Z 368.315,A -85,B 0,C 180,E1 -18200.307,E2 -18200.307} C_VEL
LIN {X 0,Y 263.212,Z 368.322,A -85,B 0,C 180,E1 -18205.291,E2 -18205.291} C_VEL
LIN {X 0,Y 263.182,Z 368.325,A -85,B 0,C 180,E1 -18208.73,E2 -18208.73} C_VEL
LIN {X 0,Y 263.169,Z 368.33,A -85,B 0,C 180,E1 -18213.193,E2 -18213.193} C_VEL
LIN {X 0,Y 263.175,Z 368.373,A -85,B 0,C 180,E1 -18214.122,E2 -18214.122} C_VEL
LIN {X 0,Y 263.62,Z 370.827,A -85,B 0,C 180,E1 -18217.819,E2 -18217.819} C_VEL
LIN {X 0,Y 264.099,Z 373.748,A -85,B 0,C 180,E1 -18221.831,E2 -18221.831} C_VEL
LIN {X 0,Y 264.596,Z 376.926,A -85,B 0,C 180,E1 -18225.82,E2 -18225.82} C_VEL
LIN {X 0,Y 264.813,Z 379.156,A -85,B 0,C 180,E1 -18228.433,E2 -18228.433} C_VEL
LIN {X 0,Y 264.861,Z 380.986,A -85,B 0,C 180,E1 -18230.444,E2 -18230.444} C_VEL
LIN {X 0,Y 264.622,Z 384.43,A -85,B 0,C 180,E1 -18233.815,E2 -18233.815} C_VEL
LIN {X 0,Y 265.775,Z 387.535,A -85,B 0,C 180,E1 -18234.126,E2 -18234.126} C_VEL
LIN {X 0,Y 269.737,Z 396.29,A -85,B 0,C 180,E1 -18235.157,E2 -18235.157} C_VEL
LIN {X 0,Y 274.269,Z 408.38,A -85,B 0,C 180,E1 -18236.604,E2 -18236.604} C_VEL
LIN {X 0,Y 277.931,Z 420.971,A -85,B 0,C 180,E1 -18238.172,E2 -18238.172} C_VEL
LIN {X 0,Y 280.479,Z 433.122,A -85,B 0,C 180,E1 -18239.786,E2 -18239.786} C_VEL
LIN {X 0,Y 281.67,Z 441.196,A -85,B 0,C 180,E1 -18240.939,E2 -18240.939} C_VEL
LIN {X 0,Y 279.355,Z 453.489,A -85,B 0,C 180,E1 -18242.466,E2 -18242.466} C_VEL
LIN {X 0,Y 276.849,Z 463.923,A -85,B 0,C 180,E1 -18244.03,E2 -18244.03} C_VEL
LIN {X 0,Y 274.347,Z 473.66,A -85,B 0,C 180,E1 -18245.803,E2 -18245.803} C_VEL
LIN {X 0,Y 271.573,Z 483.416,A -85,B 0,C 180,E1 -18247.961,E2 -18247.961} C_VEL
LIN {X 0,Y 268.834,Z 492.783,A -85,B 0,C 180,E1 -18250.544,E2 -18250.544} C_VEL
LIN {X 0,Y 266.657,Z 500.304,A -85,B 0,C 180,E1 -18253.147,E2 -18253.147} C_VEL
LIN {X 0,Y 265.043,Z 505.625,A -85,B 0,C 180,E1 -18255.41,E2 -18255.41} C_VEL
LIN {X 0,Y 263.425,Z 511.242,A -85,B 0,C 180,E1 -18258.458,E2 -18258.458} C_VEL
LIN {X 0,Y 262.56,Z 514.504,A -85,B 0,C 180,E1 -18260.758,E2 -18260.758} C_VEL
LIN {X 0,Y 261.869,Z 517.608,A -85,B 0,C 180,E1 -18263.837,E2 -18263.837} C_VEL
LIN {X 0,Y 261.434,Z 519.445,A -85,B 0,C 180,E1 -18266.918,E2 -18266.918} C_VEL
LIN {X 0,Y 261.264,Z 520.067,A -85,B 0,C 180,E1 -18270,E2 -18270} C_VEL
LIN {X 0,Y 261.432,Z 519.49,A -85,B 0,C 180,E1 -18273.082,E2 -18273.082} C_VEL
LIN {X 0,Y 261.834,Z 517.704,A -85,B 0,C 180,E1 -18276.164,E2 -18276.164} C_VEL
LIN {X 0,Y 262.556,Z 514.646,A -85,B 0,C 180,E1 -18279.242,E2 -18279.242} C_VEL
LIN {X 0,Y 263.742,Z 510.215,A -85,B 0,C 180,E1 -18282.309,E2 -18282.309} C_VEL
LIN {X 0,Y 265.407,Z 504.246,A -85,B 0,C 180,E1 -18285.355,E2 -18285.355} C_VEL
LIN {X 0,Y 267.574,Z 497.603,A -85,B 0,C 180,E1 -18287.976,E2 -18287.976} C_VEL
LIN {X 0,Y 269.853,Z 489.399,A -85,B 0,C 180,E1 -18290.584,E2 -18290.584} C_VEL
LIN {X 0,Y 272.374,Z 480.867,A -85,B 0,C 180,E1 -18292.771,E2 -18292.771} C_VEL
LIN {X 0,Y 275.196,Z 470.557,A -85,B 0,C 180,E1 -18294.922,E2 -18294.922} C_VEL
LIN {X 0,Y 277.883,Z 460.222,A -85,B 0,C 180,E1 -18296.675,E2 -18296.675} C_VEL
LIN {X 0,Y 280.364,Z 449.051,A -85,B 0,C 180,E1 -18298.239,E2 -18298.239} C_VEL
LIN {X 0,Y 281.719,Z 441.24,A -85,B 0,C 180,E1 -18299.174,E2 -18299.174} C_VEL
LIN {X 0,Y 279.956,Z 429.868,A -85,B 0,C 180,E1 -18300.78,E2 -18300.78} C_VEL
LIN {X 0,Y 276.939,Z 417.011,A -85,B 0,C 180,E1 -18302.456,E2 -18302.456} C_VEL
LIN {X 0,Y 272.659,Z 403.727,A -85,B 0,C 180,E1 -18304.089,E2 -18304.089} C_VEL
LIN {X 0,Y 267.418,Z 390.971,A -85,B 0,C 180,E1 -18305.609,E2 -18305.609} C_VEL
LIN {X 0,Y 265.723,Z 387.396,A -85,B 0,C 180,E1 -18306.023,E2 -18306.023} C_VEL
LIN {X 0,Y 264.61,Z 384.241,A -85,B 0,C 180,E1 -18306.337,E2 -18306.337} C_VEL
LIN {X 0,Y 264.866,Z 380.986,A -85,B 0,C 180,E1 -18309.691,E2 -18309.691} C_VEL
LIN {X 0,Y 264.775,Z 378.948,A -85,B 0,C 180,E1 -18311.994,E2 -18311.994} C_VEL
LIN {X 0,Y 264.393,Z 375.716,A -85,B 0,C 180,E1 -18315.866,E2 -18315.866} C_VEL
LIN {X 0,Y 264.104,Z 373.797,A -85,B 0,C 180,E1 -18318.297,E2 -18318.297} C_VEL
LIN {X 0,Y 263.646,Z 370.944,A -85,B 0,C 180,E1 -18322.185,E2 -18322.185} C_VEL
LIN {X 0,Y 263.182,Z 368.326,A -85,B 0,C 180,E1 -18326.185,E2 -18326.185} C_VEL
LIN {X 0,Y 263.154,Z 368.328,A -85,B 0,C 180,E1 -18329.507,E2 -18329.507} C_VEL
LIN {X 0,Y 263.198,Z 368.326,A -85,B 0,C 180,E1 -18333.003,E2 -18333.003} C_VEL
LIN {X 0,Y 263.188,Z 368.322,A -85,B 0,C 180,E1 -18336.387,E2 -18336.387} C_VEL
LIN {X 0,Y 263.268,Z 368.312,A -85,B 0,C 180,E1 -18339.693,E2 -18339.693} C_VEL
LIN {X 0,Y 263.355,Z 368.301,A -85,B 0,C 180,E1 -18344.522,E2 -18344.522} C_VEL
LIN {X 0,Y 263.379,Z 368.301,A -85,B 0,C 180,E1 -18349.234,E2 -18349.234} C_VEL
LIN {X 0,Y 263.578,Z 368.274,A -85,B 0,C 180,E1 -18352.338,E2 -18352.338} C_VEL
LIN {X 0,Y 263.756,Z 368.249,A -85,B 0,C 180,E1 -18358.473,E2 -18358.473} C_VEL
LIN {X 0,Y 263.755,Z 368.249,A -85,B 0,C 180,E1 -18361.527,E2 -18361.527} C_VEL
LIN {X 0,Y 263.548,Z 368.276,A -85,B 0,C 180,E1 -18367.662,E2 -18367.662} C_VEL
LIN {X 0,Y 263.359,Z 368.301,A -85,B 0,C 180,E1 -18370.766,E2 -18370.766} C_VEL
LIN {X 0,Y 263.355,Z 368.313,A -85,B 0,C 180,E1 -18375.477,E2 -18375.477} C_VEL
LIN {X 0,Y 263.35,Z 368.311,A -85,B 0,C 180,E1 -18376.053,E2 -18376.053} C_VEL
LIN {X 0,Y 262.683,Z 368.393,A -85,B 0,C 180,E1 -18377.328,E2 -18377.328} C_VEL
LIN {X 0,Y 259.763,Z 368.757,A -85,B 0,C 180,E1 -18379.404,E2 -18379.404} C_VEL
LIN {X 0,Y 257.269,Z 369.07,A -85,B 0,C 180,E1 -18381.093,E2 -18381.093} C_VEL
LIN {X 0,Y 256.195,Z 369.197,A -85,B 0,C 180,E1 -18382.405,E2 -18382.405} C_VEL
LIN {X 0,Y 256.107,Z 369.205,A -85,B 0,C 180,E1 -18382.85,E2 -18382.85} C_VEL
LIN {X 0,Y 256.172,Z 369.318,A -85,B 0,C 180,E1 -18385.768,E2 -18385.768} C_VEL
LIN {X 0,Y 256.71,Z 372.096,A -85,B 0,C 180,E1 -18389.524,E2 -18389.524} C_VEL
LIN {X 0,Y 257.272,Z 375.087,A -85,B 0,C 180,E1 -18393.116,E2 -18393.116} C_VEL
LIN {X 0,Y 257.97,Z 378.52,A -85,B 0,C 180,E1 -18396.823,E2 -18396.823} C_VEL
LIN {X 0,Y 258.744,Z 382.45,A -85,B 0,C 180,E1 -18400.684,E2 -18400.684} C_VEL
LIN {X 0,Y 259.606,Z 386.93,A -85,B 0,C 180,E1 -18404.738,E2 -18404.738} C_VEL
LIN {X 0,Y 260.195,Z 390.229,A -85,B 0,C 180,E1 -18407.525,E2 -18407.525} C_VEL
LIN {X 0,Y 260.797,Z 393.814,A -85,B 0,C 180,E1 -18410.377,E2 -18410.377} C_VEL
LIN {X 0,Y 262.127,Z 397.127,A -85,B 0,C 180,E1 -18410.729,E2 -18410.729} C_VEL
LIN {X 0,Y 263.341,Z 399.312,A -85,B 0,C 180,E1 -18411.024,E2 -18411.024} C_VEL
LIN {X 0,Y 265.765,Z 404.938,A -85,B 0,C 180,E1 -18411.675,E2 -18411.675} C_VEL
LIN {X 0,Y 269.702,Z 419.284,A -85,B 0,C 180,E1 -18413.159,E2 -18413.159} C_VEL
LIN {X 0,Y 272.396,Z 433.391,A -85,B 0,C 180,E1 -18414.718,E2 -18414.718} C_VEL
LIN {X 0,Y 274.028,Z 447.336,A -85,B 0,C 180,E1 -18416.407,E2 -18416.407} C_VEL
LIN {X 0,Y 274.554,Z 457.561,A -85,B 0,C 180,E1 -18417.775,E2 -18417.775} C_VEL
LIN {X 0,Y 271.911,Z 469.891,A -85,B 0,C 180,E1 -18419.304,E2 -18419.304} C_VEL
LIN {X 0,Y 268.596,Z 482.833,A -85,B 0,C 180,E1 -18421.262,E2 -18421.262} C_VEL
LIN {X 0,Y 265.685,Z 493.642,A -85,B 0,C 180,E1 -18423.276,E2 -18423.276} C_VEL
LIN {X 0,Y 262.773,Z 504.461,A -85,B 0,C 180,E1 -18425.743,E2 -18425.743} C_VEL
LIN {X 0,Y 260.309,Z 513.363,A -85,B 0,C 180,E1 -18428.208,E2 -18428.208} C_VEL
LIN {X 0,Y 258.057,Z 521.453,A -85,B 0,C 180,E1 -18430.924,E2 -18430.924} C_VEL
LIN {X 0,Y 256.203,Z 528.983,A -85,B 0,C 180,E1 -18434.079,E2 -18434.079} C_VEL
LIN {X 0,Y 254.984,Z 534.926,A -85,B 0,C 180,E1 -18437.261,E2 -18437.261} C_VEL
LIN {X 0,Y 254.31,Z 539.438,A -85,B 0,C 180,E1 -18440.455,E2 -18440.455} C_VEL
LIN {X 0,Y 254.05,Z 542.616,A -85,B 0,C 180,E1 -18443.647,E2 -18443.647} C_VEL
LIN {X 0,Y 254.094,Z 544.519,A -85,B 0,C 180,E1 -18446.829,E2 -18446.829} C_VEL
LIN {X 0,Y 254.17,Z 545.162,A -85,B 0,C 180,E1 -18450,E2 -18450} C_VEL
LIN {X 0,Y 254.098,Z 544.507,A -85,B 0,C 180,E1 -18453.171,E2 -18453.171} C_VEL
LIN {X 0,Y 254.115,Z 542.593,A -85,B 0,C 180,E1 -18456.351,E2 -18456.351} C_VEL
LIN {X 0,Y 254.31,Z 539.403,A -85,B 0,C 180,E1 -18459.544,E2 -18459.544} C_VEL
LIN {X 0,Y 254.982,Z 534.882,A -85,B 0,C 180,E1 -18462.738,E2 -18462.738} C_VEL
LIN {X 0,Y 256.135,Z 528.916,A -85,B 0,C 180,E1 -18465.925,E2 -18465.925} C_VEL
LIN {X 0,Y 258.055,Z 521.368,A -85,B 0,C 180,E1 -18469.075,E2 -18469.075} C_VEL
LIN {X 0,Y 260.286,Z 513.263,A -85,B 0,C 180,E1 -18471.794,E2 -18471.794} C_VEL
LIN {X 0,Y 262.798,Z 504.177,A -85,B 0,C 180,E1 -18474.3,E2 -18474.3} C_VEL
LIN {X 0,Y 265.643,Z 493.497,A -85,B 0,C 180,E1 -18476.728,E2 -18476.728} C_VEL
LIN {X 0,Y 268.597,Z 482.668,A -85,B 0,C 180,E1 -18478.737,E2 -18478.737} C_VEL
LIN {X 0,Y 271.567,Z 470.98,A -85,B 0,C 180,E1 -18480.523,E2 -18480.523} C_VEL
LIN {X 0,Y 274.433,Z 458.665,A -85,B 0,C 180,E1 -18482.055,E2 -18482.055} C_VEL
LIN {X 0,Y 273.951,Z 447.153,A -85,B 0,C 180,E1 -18483.587,E2 -18483.587} C_VEL
LIN {X 0,Y 272.393,Z 433.93,A -85,B 0,C 180,E1 -18485.192,E2 -18485.192} C_VEL
LIN {X 0,Y 269.575,Z 418.975,A -85,B 0,C 180,E1 -18486.843,E2 -18486.843} C_VEL
LIN {X 0,Y 266.152,Z 406.438,A -85,B 0,C 180,E1 -18488.14,E2 -18488.14} C_VEL
LIN {X 0,Y 263.955,Z 400.751,A -85,B 0,C 180,E1 -18488.769,E2 -18488.769} C_VEL
LIN {X 0,Y 262.523,Z 397.71,A -85,B 0,C 180,E1 -18489.133,E2 -18489.133} C_VEL
LIN {X 0,Y 260.989,Z 394.513,A -85,B 0,C 180,E1 -18489.518,E2 -18489.518} C_VEL
LIN {X 0,Y 260.785,Z 393.737,A -85,B 0,C 180,E1 -18489.586,E2 -18489.586} C_VEL
LIN {X 0,Y 260.06,Z 389.362,A -85,B 0,C 180,E1 -18493.142,E2 -18493.142} C_VEL
LIN {X 0,Y 259.141,Z 384.55,A -85,B 0,C 180,E1 -18497.312,E2 -18497.312} C_VEL
LIN {X 0,Y 258.344,Z 380.332,A -85,B 0,C 180,E1 -18501.267,E2 -18501.267} C_VEL
LIN {X 0,Y 257.613,Z 376.683,A -85,B 0,C 180,E1 -18505.047,E2 -18505.047} C_VEL
LIN {X 0,Y 256.958,Z 373.466,A -85,B 0,C 180,E1 -18508.69,E2 -18508.69} C_VEL
LIN {X 0,Y 256.497,Z 370.672,A -85,B 0,C 180,E1 -18512.238,E2 -18512.238} C_VEL
LIN {X 0,Y 256.163,Z 369.199,A -85,B 0,C 180,E1 -18514.499,E2 -18514.499} C_VEL
LIN {X 0,Y 256.169,Z 369.195,A -85,B 0,C 180,E1 -18519.105,E2 -18519.105} C_VEL
LIN {X 0,Y 256.302,Z 369.176,A -85,B 0,C 180,E1 -18524.085,E2 -18524.085} C_VEL
LIN {X 0,Y 256.298,Z 369.177,A -85,B 0,C 180,E1 -18527.328,E2 -18527.328} C_VEL
LIN {X 0,Y 256.508,Z 369.159,A -85,B 0,C 180,E1 -18532.126,E2 -18532.126} C_VEL
LIN {X 0,Y 256.501,Z 369.151,A -85,B 0,C 180,E1 -18536.859,E2 -18536.859} C_VEL
LIN {X 0,Y 256.768,Z 369.119,A -85,B 0,C 180,E1 -18540,E2 -18540} C_VEL
LIN {X 0,Y 256.502,Z 369.156,A -85,B 0,C 180,E1 -18543.142,E2 -18543.142} C_VEL
LIN {X 0,Y 256.544,Z 369.145,A -85,B 0,C 180,E1 -18547.873,E2 -18547.873} C_VEL
LIN {X 0,Y 256.314,Z 369.175,A -85,B 0,C 180,E1 -18551.066,E2 -18551.066} C_VEL
LIN {X 0,Y 256.303,Z 369.181,A -85,B 0,C 180,E1 -18555.915,E2 -18555.915} C_VEL
LIN {X 0,Y 256.17,Z 369.195,A -85,B 0,C 180,E1 -18560.895,E2 -18560.895} C_VEL
LIN {X 0,Y 256.191,Z 369.195,A -85,B 0,C 180,E1 -18565.139,E2 -18565.139} C_VEL
LIN {X 0,Y 256.117,Z 369.201,A -85,B 0,C 180,E1 -18569.6,E2 -18569.6} C_VEL
LIN {X 0,Y 256.133,Z 369.295,A -85,B 0,C 180,E1 -18572.806,E2 -18572.806} C_VEL
LIN {X 0,Y 256.695,Z 372.217,A -85,B 0,C 180,E1 -18577.44,E2 -18577.44} C_VEL
LIN {X 0,Y 257.057,Z 374.731,A -85,B 0,C 180,E1 -18581.009,E2 -18581.009} C_VEL
LIN {X 0,Y 257.555,Z 377.917,A -85,B 0,C 180,E1 -18585.192,E2 -18585.192} C_VEL
LIN {X 0,Y 257.788,Z 379.725,A -85,B 0,C 180,E1 -18587.4,E2 -18587.4} C_VEL
LIN {X 0,Y 257.819,Z 383.08,A -85,B 0,C 180,E1 -18591.173,E2 -18591.173} C_VEL
LIN {X 0,Y 257.727,Z 384.439,A -85,B 0,C 180,E1 -18592.61,E2 -18592.61} C_VEL
LIN {X 0,Y 258.927,Z 387.671,A -85,B 0,C 180,E1 -18592.962,E2 -18592.962} C_VEL
LIN {X 0,Y 261.82,Z 393.79,A -85,B 0,C 180,E1 -18593.737,E2 -18593.737} C_VEL
LIN {X 0,Y 266.884,Z 406.318,A -85,B 0,C 180,E1 -18595.325,E2 -18595.325} C_VEL
LIN {X 0,Y 270.799,Z 419.116,A -85,B 0,C 180,E1 -18596.975,E2 -18596.975} C_VEL
LIN {X 0,Y 273.621,Z 431.386,A -85,B 0,C 180,E1 -18598.66,E2 -18598.66} C_VEL
LIN {X 0,Y 275.218,Z 442.192,A -85,B 0,C 180,E1 -18600.254,E2 -18600.254} C_VEL
LIN {X 0,Y 274.974,Z 445.027,A -85,B 0,C 180,E1 -18600.622,E2 -18600.622} C_VEL
LIN {X 0,Y 272.514,Z 456.445,A -85,B 0,C 180,E1 -18602.132,E2 -18602.132} C_VEL
LIN {X 0,Y 269.911,Z 466.471,A -85,B 0,C 180,E1 -18603.727,E2 -18603.727} C_VEL
LIN {X 0,Y 267.41,Z 475.82,A -85,B 0,C 180,E1 -18605.548,E2 -18605.548} C_VEL
LIN {X 0,Y 264.565,Z 485.26,A -85,B 0,C 180,E1 -18607.757,E2 -18607.757} C_VEL
LIN {X 0,Y 261.841,Z 494.313,A -85,B 0,C 180,E1 -18610.396,E2 -18610.396} C_VEL
LIN {X 0,Y 259.888,Z 500.662,A -85,B 0,C 180,E1 -18612.694,E2 -18612.694} C_VEL
LIN {X 0,Y 258.15,Z 505.98,A -85,B 0,C 180,E1 -18615.011,E2 -18615.011} C_VEL
LIN {X 0,Y 256.453,Z 511.593,A -85,B 0,C 180,E1 -18618.139,E2 -18618.139} C_VEL
LIN {X 0,Y 255.564,Z 514.852,A -85,B 0,C 180,E1 -18620.503,E2 -18620.503} C_VEL
LIN {X 0,Y 254.807,Z 517.955,A -85,B 0,C 180,E1 -18623.666,E2 -18623.666} C_VEL
LIN {X 0,Y 254.371,Z 519.789,A -85,B 0,C 180,E1 -18626.832,E2 -18626.832} C_VEL
LIN {X 0,Y 254.186,Z 520.411,A -85,B 0,C 180,E1 -18630,E2 -18630} C_VEL
LIN {X 0,Y 254.369,Z 519.834,A -85,B 0,C 180,E1 -18633.168,E2 -18633.168} C_VEL
LIN {X 0,Y 254.771,Z 518.049,A -85,B 0,C 180,E1 -18636.335,E2 -18636.335} C_VEL
LIN {X 0,Y 255.561,Z 514.992,A -85,B 0,C 180,E1 -18639.498,E2 -18639.498} C_VEL
LIN {X 0,Y 256.795,Z 510.564,A -85,B 0,C 180,E1 -18642.647,E2 -18642.647} C_VEL
LIN {X 0,Y 258.555,Z 504.599,A -85,B 0,C 180,E1 -18645.773,E2 -18645.773} C_VEL
LIN {X 0,Y 260.836,Z 497.961,A -85,B 0,C 180,E1 -18648.457,E2 -18648.457} C_VEL
LIN {X 0,Y 263.222,Z 489.767,A -85,B 0,C 180,E1 -18651.127,E2 -18651.127} C_VEL
LIN {X 0,Y 265.859,Z 481.247,A -85,B 0,C 180,E1 -18653.362,E2 -18653.362} C_VEL
LIN {X 0,Y 268.785,Z 470.956,A -85,B 0,C 180,E1 -18655.559,E2 -18655.559} C_VEL
LIN {X 0,Y 271.576,Z 460.647,A -85,B 0,C 180,E1 -18657.345,E2 -18657.345} C_VEL
LIN {X 0,Y 274.453,Z 448.086,A -85,B 0,C 180,E1 -18659.114,E2 -18659.114} C_VEL
LIN {X 0,Y 275.337,Z 442.701,A -85,B 0,C 180,E1 -18659.789,E2 -18659.789} C_VEL
LIN {X 0,Y 273.802,Z 432.111,A -85,B 0,C 180,E1 -18661.357,E2 -18661.357} C_VEL
LIN {X 0,Y 270.817,Z 418.813,A -85,B 0,C 180,E1 -18663.183,E2 -18663.183} C_VEL
LIN {X 0,Y 266.487,Z 405.181,A -85,B 0,C 180,E1 -18664.956,E2 -18664.956} C_VEL
LIN {X 0,Y 261.031,Z 391.884,A -85,B 0,C 180,E1 -18666.634,E2 -18666.634} C_VEL
LIN {X 0,Y 258.753,Z 387.315,A -85,B 0,C 180,E1 -18667.222,E2 -18667.222} C_VEL
LIN {X 0,Y 257.743,Z 384.398,A -85,B 0,C 180,E1 -18667.569,E2 -18667.569} C_VEL
LIN {X 0,Y 257.843,Z 381.367,A -85,B 0,C 180,E1 -18670.857,E2 -18670.857} C_VEL
LIN {X 0,Y 257.572,Z 378.074,A -85,B 0,C 180,E1 -18674.811,E2 -18674.811} C_VEL
LIN {X 0,Y 257.079,Z 374.864,A -85,B 0,C 180,E1 -18678.996,E2 -18678.996} C_VEL
LIN {X 0,Y 256.658,Z 372.077,A -85,B 0,C 180,E1 -18682.956,E2 -18682.956} C_VEL
LIN {X 0,Y 256.118,Z 369.277,A -85,B 0,C 180,E1 -18687.43,E2 -18687.43} C_VEL
LIN {X 0,Y 256.146,Z 369.202,A -85,B 0,C 180,E1 -18692.196,E2 -18692.196} C_VEL
LIN {X 0,Y 256.171,Z 369.199,A -85,B 0,C 180,E1 -18695.699,E2 -18695.699} C_VEL
LIN {X 0,Y 256.171,Z 369.195,A -85,B 0,C 180,E1 -18699.105,E2 -18699.105} C_VEL
LIN {X 0,Y 256.304,Z 369.182,A -85,B 0,C 180,E1 -18704.085,E2 -18704.085} C_VEL
LIN {X 0,Y 256.314,Z 369.178,A -85,B 0,C 180,E1 -18708.934,E2 -18708.934} C_VEL
LIN {X 0,Y 256.545,Z 369.149,A -85,B 0,C 180,E1 -18712.127,E2 -18712.127} C_VEL
LIN {X 0,Y 256.719,Z 369.125,A -85,B 0,C 180,E1 -18718.431,E2 -18718.431} C_VEL
LIN {X 0,Y 256.718,Z 369.125,A -85,B 0,C 180,E1 -18721.568,E2 -18721.568} C_VEL
LIN {X 0,Y 256.479,Z 369.163,A -85,B 0,C 180,E1 -18726.292,E2 -18726.292} C_VEL
LIN {X 0,Y 256.43,Z 369.171,A -85,B 0,C 180,E1 -18729.465,E2 -18729.465} C_VEL
LIN {X 0,Y 256.26,Z 369.188,A -85,B 0,C 180,E1 -18734.29,E2 -18734.29} C_VEL
LIN {X 0,Y 256.215,Z 369.196,A -85,B 0,C 180,E1 -18737.561,E2 -18737.561} C_VEL
LIN {X 0,Y 256.189,Z 369.205,A -85,B 0,C 180,E1 -18741.136,E2 -18741.136} C_VEL
LIN {X 0,Y 256.107,Z 369.205,A -85,B 0,C 180,E1 -18742.85,E2 -18742.85} C_VEL
LIN {X 0,Y 255.495,Z 369.521,A -85,B 0,C 180,E1 -18744.16,E2 -18744.16} C_VEL
LIN {X 0,Y 252.927,Z 371.046,A -85,B 0,C 180,E1 -18746.288,E2 -18746.288} C_VEL
LIN {X 0,Y 250.794,Z 372.697,A -85,B 0,C 180,E1 -18748.008,E2 -18748.008} C_VEL
LIN {X 0,Y 249.947,Z 373.914,A -85,B 0,C 180,E1 -18749.335,E2 -18749.335} C_VEL
LIN {X 0,Y 249.913,Z 374.279,A -85,B 0,C 180,E1 -18749.784,E2 -18749.784} C_VEL
LIN {X 0,Y 250.597,Z 377.864,A -85,B 0,C 180,E1 -18754.118,E2 -18754.118} C_VEL
LIN {X 0,Y 251.444,Z 381.938,A -85,B 0,C 180,E1 -18758.498,E2 -18758.498} C_VEL
LIN {X 0,Y 252.109,Z 385.533,A -85,B 0,C 180,E1 -18761.993,E2 -18761.993} C_VEL
LIN {X 0,Y 252.993,Z 390.217,A -85,B 0,C 180,E1 -18766.241,E2 -18766.241} C_VEL
LIN {X 0,Y 253.588,Z 393.66,A -85,B 0,C 180,E1 -18769.081,E2 -18769.081} C_VEL
LIN {X 0,Y 254.949,Z 396.943,A -85,B 0,C 180,E1 -18769.462,E2 -18769.462} C_VEL
LIN {X 0,Y 256.437,Z 399.613,A -85,B 0,C 180,E1 -18769.846,E2 -18769.846} C_VEL
LIN {X 0,Y 259.982,Z 407.137,A -85,B 0,C 180,E1 -18770.839,E2 -18770.839} C_VEL
LIN {X 0,Y 263.281,Z 419.05,A -85,B 0,C 180,E1 -18772.153,E2 -18772.153} C_VEL
LIN {X 0,Y 265.958,Z 433.079,A -85,B 0,C 180,E1 -18773.767,E2 -18773.767} C_VEL
LIN {X 0,Y 267.634,Z 446.929,A -85,B 0,C 180,E1 -18775.513,E2 -18775.513} C_VEL
LIN {X 0,Y 268.151,Z 457.707,A -85,B 0,C 180,E1 -18777.002,E2 -18777.002} C_VEL
LIN {X 0,Y 267.809,Z 461.081,A -85,B 0,C 180,E1 -18777.44,E2 -18777.44} C_VEL
LIN {X 0,Y 264.468,Z 474.478,A -85,B 0,C 180,E1 -18779.232,E2 -18779.232} C_VEL
LIN {X 0,Y 261.443,Z 485.598,A -85,B 0,C 180,E1 -18781.061,E2 -18781.061} C_VEL
LIN {X 0,Y 258.272,Z 496.801,A -85,B 0,C 180,E1 -18783.321,E2 -18783.321} C_VEL
LIN {X 0,Y 255.608,Z 506.255,A -85,B 0,C 180,E1 -18785.642,E2 -18785.642} C_VEL
LIN {X 0,Y 252.879,Z 515.502,A -85,B 0,C 180,E1 -18788.392,E2 -18788.392} C_VEL
LIN {X 0,Y 250.733,Z 523.161,A -85,B 0,C 180,E1 -18791.195,E2 -18791.195} C_VEL
LIN {X 0,Y 248.931,Z 530.292,A -85,B 0,C 180,E1 -18794.442,E2 -18794.442} C_VEL
LIN {X 0,Y 247.727,Z 535.863,A -85,B 0,C 180,E1 -18797.715,E2 -18797.715} C_VEL
LIN {X 0,Y 247.262,Z 539.09,A -85,B 0,C 180,E1 -18800.181,E2 -18800.181} C_VEL
LIN {X 0,Y 246.962,Z 542.269,A -85,B 0,C 180,E1 -18803.464,E2 -18803.464} C_VEL
LIN {X 0,Y 246.989,Z 543.38,A -85,B 0,C 180,E1 -18805.103,E2 -18805.103} C_VEL
LIN {X 0,Y 247.062,Z 544.655,A -85,B 0,C 180,E1 -18808.37,E2 -18808.37} C_VEL
LIN {X 0,Y 247.094,Z 544.818,A -85,B 0,C 180,E1 -18810,E2 -18810} C_VEL
LIN {X 0,Y 247.011,Z 544.162,A -85,B 0,C 180,E1 -18813.262,E2 -18813.262} C_VEL
LIN {X 0,Y 247.026,Z 542.245,A -85,B 0,C 180,E1 -18816.534,E2 -18816.534} C_VEL
LIN {X 0,Y 247.262,Z 539.053,A -85,B 0,C 180,E1 -18819.819,E2 -18819.819} C_VEL
LIN {X 0,Y 247.974,Z 534.528,A -85,B 0,C 180,E1 -18823.105,E2 -18823.105} C_VEL
LIN {X 0,Y 249.364,Z 528.071,A -85,B 0,C 180,E1 -18826.616,E2 -18826.616} C_VEL
LIN {X 0,Y 251.542,Z 519.967,A -85,B 0,C 180,E1 -18830.015,E2 -18830.015} C_VEL
LIN {X 0,Y 254.03,Z 511.636,A -85,B 0,C 180,E1 -18832.788,E2 -18832.788} C_VEL
LIN {X 0,Y 256.857,Z 501.694,A -85,B 0,C 180,E1 -18835.502,E2 -18835.502} C_VEL
LIN {X 0,Y 259.78,Z 491.296,A -85,B 0,C 180,E1 -18837.819,E2 -18837.819} C_VEL
LIN {X 0,Y 263.171,Z 478.994,A -85,B 0,C 180,E1 -18840.048,E2 -18840.048} C_VEL
LIN {X 0,Y 266.446,Z 466.627,A -85,B 0,C 180,E1 -18841.839,E2 -18841.839} C_VEL
LIN {X 0,Y 268.109,Z 459.62,A -85,B 0,C 180,E1 -18842.699,E2 -18842.699} C_VEL
LIN {X 0,Y 267.592,Z 446.895,A -85,B 0,C 180,E1 -18844.457,E2 -18844.457} C_VEL
LIN {X 0,Y 266.031,Z 433.93,A -85,B 0,C 180,E1 -18846.094,E2 -18846.094} C_VEL
LIN {X 0,Y 263.475,Z 420.309,A -85,B 0,C 180,E1 -18847.674,E2 -18847.674} C_VEL
LIN {X 0,Y 260.166,Z 407.813,A -85,B 0,C 180,E1 -18849.046,E2 -18849.046} C_VEL
LIN {X 0,Y 257.328,Z 401.419,A -85,B 0,C 180,E1 -18849.869,E2 -18849.869} C_VEL
LIN {X 0,Y 255.502,Z 397.807,A -85,B 0,C 180,E1 -18850.35,E2 -18850.35} C_VEL
LIN {X 0,Y 253.825,Z 394.535,A -85,B 0,C 180,E1 -18850.791,E2 -18850.791} C_VEL
LIN {X 0,Y 253.556,Z 393.498,A -85,B 0,C 180,E1 -18850.91,E2 -18850.91} C_VEL
LIN {X 0,Y 252.762,Z 388.77,A -85,B 0,C 180,E1 -18854.969,E2 -18854.969} C_VEL
LIN {X 0,Y 251.932,Z 384.529,A -85,B 0,C 180,E1 -18858.869,E2 -18858.869} C_VEL
LIN {X 0,Y 251.323,Z 381.35,A -85,B 0,C 180,E1 -18862.033,E2 -18862.033} C_VEL
LIN {X 0,Y 250.586,Z 377.791,A -85,B 0,C 180,E1 -18865.881,E2 -18865.881} C_VEL
LIN {X 0,Y 249.982,Z 374.689,A -85,B 0,C 180,E1 -18869.599,E2 -18869.599} C_VEL
LIN {X 0,Y 249.802,Z 373.263,A -85,B 0,C 180,E1 -18871.427,E2 -18871.427} C_VEL
LIN {X 0,Y 249.096,Z 370.079,A -85,B 0,C 180,E1 -18876.073,E2 -18876.073} C_VEL
LIN {X 0,Y 249.114,Z 370.08,A -85,B 0,C 180,E1 -18880.212,E2 -18880.212} C_VEL
LIN {X 0,Y 249.244,Z 370.057,A -85,B 0,C 180,E1 -18883.622,E2 -18883.622} C_VEL
LIN {X 0,Y 249.247,Z 370.064,A -85,B 0,C 180,E1 -18888.617,E2 -18888.617} C_VEL
LIN {X 0,Y 249.449,Z 370.039,A -85,B 0,C 180,E1 -18891.902,E2 -18891.902} C_VEL
LIN {X 0,Y 249.298,Z 370.058,A -85,B 0,C 180,E1 -18895.149,E2 -18895.149} C_VEL
LIN {X 0,Y 249.679,Z 370.008,A -85,B 0,C 180,E1 -18898.387,E2 -18898.387} C_VEL
LIN {X 0,Y 249.679,Z 370.004,A -85,B 0,C 180,E1 -18901.613,E2 -18901.613} C_VEL
LIN {X 0,Y 249.454,Z 370.033,A -85,B 0,C 180,E1 -18906.773,E2 -18906.773} C_VEL
LIN {X 0,Y 249.427,Z 370.042,A -85,B 0,C 180,E1 -18909.733,E2 -18909.733} C_VEL
LIN {X 0,Y 249.209,Z 370.06,A -85,B 0,C 180,E1 -18914.703,E2 -18914.703} C_VEL
LIN {X 0,Y 249.143,Z 370.069,A -85,B 0,C 180,E1 -18918.077,E2 -18918.077} C_VEL
LIN {X 0,Y 249.09,Z 370.076,A -85,B 0,C 180,E1 -18921.518,E2 -18921.518} C_VEL
LIN {X 0,Y 249.134,Z 370.078,A -85,B 0,C 180,E1 -18925.482,E2 -18925.482} C_VEL
LIN {X 0,Y 249.086,Z 370.078,A -85,B 0,C 180,E1 -18928.994,E2 -18928.994} C_VEL
LIN {X 0,Y 249.079,Z 370.231,A -85,B 0,C 180,E1 -18931.366,E2 -18931.366} C_VEL
LIN {X 0,Y 249.519,Z 372.481,A -85,B 0,C 180,E1 -18935.232,E2 -18935.232} C_VEL
LIN {X 0,Y 249.839,Z 374.404,A -85,B 0,C 180,E1 -18938.234,E2 -18938.234} C_VEL
LIN {X 0,Y 250.306,Z 377.305,A -85,B 0,C 180,E1 -18942.366,E2 -18942.366} C_VEL
LIN {X 0,Y 250.779,Z 380.7,A -85,B 0,C 180,E1 -18946.773,E2 -18946.773} C_VEL
LIN {X 0,Y 250.904,Z 383.342,A -85,B 0,C 180,E1 -18949.891,E2 -18949.891} C_VEL
LIN {X 0,Y 250.864,Z 384.818,A -85,B 0,C 180,E1 -18951.357,E2 -18951.357} C_VEL
LIN {X 0,Y 252.104,Z 387.989,A -85,B 0,C 180,E1 -18951.727,E2 -18951.727} C_VEL
LIN {X 0,Y 253.312,Z 390.153,A -85,B 0,C 180,E1 -18952.044,E2 -18952.044} C_VEL
LIN {X 0,Y 258.564,Z 402.051,A -85,B 0,C 180,E1 -18953.658,E2 -18953.658} C_VEL
LIN {X 0,Y 262.82,Z 414.323,A -85,B 0,C 180,E1 -18955.314,E2 -18955.314} C_VEL
LIN {X 0,Y 266.024,Z 426.467,A -85,B 0,C 180,E1 -18957.013,E2 -18957.013} C_VEL
LIN {X 0,Y 268.037,Z 437.119,A -85,B 0,C 180,E1 -18958.591,E2 -18958.591} C_VEL
LIN {X 0,Y 268.943,Z 444.804,A -85,B 0,C 180,E1 -18959.79,E2 -18959.79} C_VEL
LIN {X 0,Y 266.284,Z 456.878,A -85,B 0,C 180,E1 -18961.421,E2 -18961.421} C_VEL
LIN {X 0,Y 263.578,Z 466.887,A -85,B 0,C 180,E1 -18963.045,E2 -18963.045} C_VEL
LIN {X 0,Y 260.974,Z 476.215,A -85,B 0,C 180,E1 -18964.903,E2 -18964.903} C_VEL
LIN {X 0,Y 258.01,Z 485.638,A -85,B 0,C 180,E1 -18967.16,E2 -18967.16} C_VEL
LIN {X 0,Y 255.45,Z 493.515,A -85,B 0,C 180,E1 -18969.478,E2 -18969.478} C_VEL
LIN {X 0,Y 253.116,Z 501.021,A -85,B 0,C 180,E1 -18972.216,E2 -18972.216} C_VEL
LIN {X 0,Y 251.282,Z 506.333,A -85,B 0,C 180,E1 -18974.591,E2 -18974.591} C_VEL
LIN {X 0,Y 249.501,Z 511.942,A -85,B 0,C 180,E1 -18977.804,E2 -18977.804} C_VEL
LIN {X 0,Y 248.548,Z 515.201,A -85,B 0,C 180,E1 -18980.232,E2 -18980.232} C_VEL
LIN {X 0,Y 247.759,Z 518.301,A -85,B 0,C 180,E1 -18983.485,E2 -18983.485} C_VEL
LIN {X 0,Y 247.309,Z 520.134,A -85,B 0,C 180,E1 -18986.742,E2 -18986.742} C_VEL
LIN {X 0,Y 247.111,Z 520.756,A -85,B 0,C 180,E1 -18990,E2 -18990} C_VEL
LIN {X 0,Y 247.308,Z 520.178,A -85,B 0,C 180,E1 -18993.258,E2 -18993.258} C_VEL
LIN {X 0,Y 247.713,Z 518.394,A -85,B 0,C 180,E1 -18996.517,E2 -18996.517} C_VEL
LIN {X 0,Y 248.543,Z 515.338,A -85,B 0,C 180,E1 -18999.768,E2 -18999.768} C_VEL
LIN {X 0,Y 249.871,Z 510.912,A -85,B 0,C 180,E1 -19003.004,E2 -19003.004} C_VEL
LIN {X 0,Y 251.72,Z 504.953,A -85,B 0,C 180,E1 -19006.213,E2 -19006.213} C_VEL
LIN {X 0,Y 254.119,Z 498.32,A -85,B 0,C 180,E1 -19008.964,E2 -19008.964} C_VEL
LIN {X 0,Y 256.615,Z 490.132,A -85,B 0,C 180,E1 -19011.699,E2 -19011.699} C_VEL
LIN {X 0,Y 259.378,Z 481.627,A -85,B 0,C 180,E1 -19013.981,E2 -19013.981} C_VEL
LIN {X 0,Y 262.412,Z 471.355,A -85,B 0,C 180,E1 -19016.226,E2 -19016.226} C_VEL
LIN {X 0,Y 265.304,Z 461.073,A -85,B 0,C 180,E1 -19018.048,E2 -19018.048} C_VEL
LIN {X 0,Y 268.29,Z 448.549,A -85,B 0,C 180,E1 -19019.849,E2 -19019.849} C_VEL
LIN {X 0,Y 269.006,Z 444.08,A -85,B 0,C 180,E1 -19020.44,E2 -19020.44} C_VEL
LIN {X 0,Y 267.194,Z 431.854,A -85,B 0,C 180,E1 -19022.329,E2 -19022.329} C_VEL
LIN {X 0,Y 264.782,Z 421.05,A -85,B 0,C 180,E1 -19023.876,E2 -19023.876} C_VEL
LIN {X 0,Y 260.793,Z 408.007,A -85,B 0,C 180,E1 -19025.673,E2 -19025.673} C_VEL
LIN {X 0,Y 255.987,Z 395.921,A -85,B 0,C 180,E1 -19027.311,E2 -19027.311} C_VEL
LIN {X 0,Y 252.525,Z 388.59,A -85,B 0,C 180,E1 -19028.311,E2 -19028.311} C_VEL
LIN {X 0,Y 250.995,Z 385.351,A -85,B 0,C 180,E1 -19028.739,E2 -19028.739} C_VEL
LIN {X 0,Y 250.872,Z 384.607,A -85,B 0,C 180,E1 -19028.827,E2 -19028.827} C_VEL
LIN {X 0,Y 250.808,Z 381.633,A -85,B 0,C 180,E1 -19032.262,E2 -19032.262} C_VEL
LIN {X 0,Y 250.556,Z 379.087,A -85,B 0,C 180,E1 -19035.473,E2 -19035.473} C_VEL
LIN {X 0,Y 250.073,Z 375.939,A -85,B 0,C 180,E1 -19039.73,E2 -19039.73} C_VEL
LIN {X 0,Y 249.647,Z 373.241,A -85,B 0,C 180,E1 -19043.758,E2 -19043.758} C_VEL
LIN {X 0,Y 249.19,Z 370.819,A -85,B 0,C 180,E1 -19047.791,E2 -19047.791} C_VEL
LIN {X 0,Y 249.056,Z 370.084,A -85,B 0,C 180,E1 -19049.473,E2 -19049.473} C_VEL
LIN {X 0,Y 249.078,Z 370.083,A -85,B 0,C 180,E1 -19053.162,E2 -19053.162} C_VEL
LIN {X 0,Y 249.084,Z 370.079,A -85,B 0,C 180,E1 -19056.733,E2 -19056.733} C_VEL
LIN {X 0,Y 249.116,Z 370.079,A -85,B 0,C 180,E1 -19060.212,E2 -19060.212} C_VEL
LIN {X 0,Y 249.246,Z 370.064,A -85,B 0,C 180,E1 -19063.622,E2 -19063.622} C_VEL
LIN {X 0,Y 249.258,Z 370.055,A -85,B 0,C 180,E1 -19068.616,E2 -19068.616} C_VEL
LIN {X 0,Y 249.489,Z 370.026,A -85,B 0,C 180,E1 -19071.903,E2 -19071.903} C_VEL
LIN {X 0,Y 249.441,Z 370.039,A -85,B 0,C 180,E1 -19076.769,E2 -19076.769} C_VEL
LIN {X 0,Y 249.733,Z 370.004,A -85,B 0,C 180,E1 -19080,E2 -19080} C_VEL
LIN {X 0,Y 249.438,Z 370.041,A -85,B 0,C 180,E1 -19083.23,E2 -19083.23} C_VEL
LIN {X 0,Y 249.451,Z 370.04,A -85,B 0,C 180,E1 -19086.47,E2 -19086.47} C_VEL
LIN {X 0,Y 249.348,Z 370.054,A -85,B 0,C 180,E1 -19089.736,E2 -19089.736} C_VEL
LIN {X 0,Y 249.21,Z 370.068,A -85,B 0,C 180,E1 -19094.703,E2 -19094.703} C_VEL
LIN {X 0,Y 249.144,Z 370.081,A -85,B 0,C 180,E1 -19098.077,E2 -19098.077} C_VEL
LIN {X 0,Y 249.107,Z 370.085,A -85,B 0,C 180,E1 -19101.516,E2 -19101.516} C_VEL
LIN {X 0,Y 249.139,Z 370.287,A -85,B 0,C 180,E1 -19104.144,E2 -19104.144} C_VEL
LIN {X 0,Y 249.798,Z 373.349,A -85,B 0,C 180,E1 -19108.574,E2 -19108.574} C_VEL
LIN {X 0,Y 249.913,Z 374.279,A -85,B 0,C 180,E1 -19109.784,E2 -19109.784} C_VEL
LIN {X 0,Y 249.433,Z 375.505,A -85,B 0,C 180,E1 -19111.103,E2 -19111.103} C_VEL
LIN {X 0,Y 247.029,Z 378.041,A -85,B 0,C 180,E1 -19113.241,E2 -19113.241} C_VEL
LIN {X 0,Y 244.998,Z 380.178,A -85,B 0,C 180,E1 -19114.973,E2 -19114.973} C_VEL
LIN {X 0,Y 244.218,Z 381.646,A -85,B 0,C 180,E1 -19116.315,E2 -19116.315} C_VEL
LIN {X 0,Y 244.206,Z 382.084,A -85,B 0,C 180,E1 -19116.77,E2 -19116.77} C_VEL
LIN {X 0,Y 244.874,Z 385.37,A -85,B 0,C 180,E1 -19120.222,E2 -19120.222} C_VEL
LIN {X 0,Y 245.695,Z 389.642,A -85,B 0,C 180,E1 -19124.347,E2 -19124.347} C_VEL
LIN {X 0,Y 246.331,Z 393.343,A -85,B 0,C 180,E1 -19127.667,E2 -19127.667} C_VEL
LIN {X 0,Y 247.636,Z 396.664,A -85,B 0,C 180,E1 -19128.065,E2 -19128.065} C_VEL
LIN {X 0,Y 249.116,Z 399.042,A -85,B 0,C 180,E1 -19128.462,E2 -19128.462} C_VEL
LIN {X 0,Y 253.511,Z 407.919,A -85,B 0,C 180,E1 -19129.75,E2 -19129.75} C_VEL
LIN {X 0,Y 255.389,Z 412.866,A -85,B 0,C 180,E1 -19130.401,E2 -19130.401} C_VEL
LIN {X 0,Y 258.369,Z 425.409,A -85,B 0,C 180,E1 -19131.876,E2 -19131.876} C_VEL
LIN {X 0,Y 260.621,Z 440.296,A -85,B 0,C 180,E1 -19133.736,E2 -19133.736} C_VEL
LIN {X 0,Y 261.642,Z 452.437,A -85,B 0,C 180,E1 -19135.399,E2 -19135.399} C_VEL
LIN {X 0,Y 261.771,Z 460.437,A -85,B 0,C 180,E1 -19136.564,E2 -19136.564} C_VEL
LIN {X 0,Y 258.714,Z 472.865,A -85,B 0,C 180,E1 -19138.242,E2 -19138.242} C_VEL
LIN {X 0,Y 255.218,Z 485.196,A -85,B 0,C 180,E1 -19140.286,E2 -19140.286} C_VEL
LIN {X 0,Y 251.878,Z 496.415,A -85,B 0,C 180,E1 -19142.587,E2 -19142.587} C_VEL
LIN {X 0,Y 249.08,Z 505.877,A -85,B 0,C 180,E1 -19144.96,E2 -19144.96} C_VEL
LIN {X 0,Y 246.231,Z 515.136,A -85,B 0,C 180,E1 -19147.778,E2 -19147.778} C_VEL
LIN {X 0,Y 243.919,Z 522.799,A -85,B 0,C 180,E1 -19150.649,E2 -19150.649} C_VEL
LIN {X 0,Y 242.013,Z 529.936,A -85,B 0,C 180,E1 -19153.985,E2 -19153.985} C_VEL
LIN {X 0,Y 240.721,Z 535.511,A -85,B 0,C 180,E1 -19157.351,E2 -19157.351} C_VEL
LIN {X 0,Y 240.19,Z 538.739,A -85,B 0,C 180,E1 -19159.888,E2 -19159.888} C_VEL
LIN {X 0,Y 239.879,Z 541.922,A -85,B 0,C 180,E1 -19163.27,E2 -19163.27} C_VEL
LIN {X 0,Y 239.924,Z 543.828,A -85,B 0,C 180,E1 -19166.641,E2 -19166.641} C_VEL
LIN {X 0,Y 240.02,Z 544.473,A -85,B 0,C 180,E1 -19170,E2 -19170} C_VEL
LIN {X 0,Y 239.989,Z 544.306,A -85,B 0,C 180,E1 -19171.678,E2 -19171.678} C_VEL
LIN {X 0,Y 239.911,Z 542.971,A -85,B 0,C 180,E1 -19175.127,E2 -19175.127} C_VEL
LIN {X 0,Y 240.004,Z 540.461,A -85,B 0,C 180,E1 -19178.419,E2 -19178.419} C_VEL
LIN {X 0,Y 240.473,Z 536.608,A -85,B 0,C 180,E1 -19181.805,E2 -19181.805} C_VEL
LIN {X 0,Y 241.584,Z 531.375,A -85,B 0,C 180,E1 -19185.178,E2 -19185.178} C_VEL
LIN {X 0,Y 243.377,Z 524.633,A -85,B 0,C 180,E1 -19188.521,E2 -19188.521} C_VEL
LIN {X 0,Y 245.439,Z 517.335,A -85,B 0,C 180,E1 -19191.413,E2 -19191.413} C_VEL
LIN {X 0,Y 248.222,Z 508.545,A -85,B 0,C 180,E1 -19194.239,E2 -19194.239} C_VEL
LIN {X 0,Y 250.881,Z 499.574,A -85,B 0,C 180,E1 -19196.629,E2 -19196.629} C_VEL
LIN {X 0,Y 254.001,Z 488.963,A -85,B 0,C 180,E1 -19198.961,E2 -19198.961} C_VEL
LIN {X 0,Y 257.317,Z 477.383,A -85,B 0,C 180,E1 -19201.033,E2 -19201.033} C_VEL
LIN {X 0,Y 260.774,Z 464.752,A -85,B 0,C 180,E1 -19202.843,E2 -19202.843} C_VEL
LIN {X 0,Y 261.777,Z 460.521,A -85,B 0,C 180,E1 -19203.382,E2 -19203.382} C_VEL
LIN {X 0,Y 261.222,Z 446.913,A -85,B 0,C 180,E1 -19205.343,E2 -19205.343} C_VEL
LIN {X 0,Y 259.576,Z 432.905,A -85,B 0,C 180,E1 -19207.176,E2 -19207.176} C_VEL
LIN {X 0,Y 256.74,Z 418.383,A -85,B 0,C 180,E1 -19208.928,E2 -19208.928} C_VEL
LIN {X 0,Y 254.092,Z 409.231,A -85,B 0,C 180,E1 -19210.021,E2 -19210.021} C_VEL
LIN {X 0,Y 250.361,Z 401.531,A -85,B 0,C 180,E1 -19211.135,E2 -19211.135} C_VEL
LIN {X 0,Y 248.264,Z 397.545,A -85,B 0,C 180,E1 -19211.717,E2 -19211.717} C_VEL
LIN {X 0,Y 246.598,Z 394.355,A -85,B 0,C 180,E1 -19212.184,E2 -19212.184} C_VEL
LIN {X 0,Y 246.33,Z 393.32,A -85,B 0,C 180,E1 -19212.289,E2 -19212.289} C_VEL
LIN {X 0,Y 245.694,Z 389.572,A -85,B 0,C 180,E1 -19215.653,E2 -19215.653} C_VEL
LIN {X 0,Y 244.872,Z 385.296,A -85,B 0,C 180,E1 -19219.777,E2 -19219.777} C_VEL
LIN {X 0,Y 244.134,Z 381.564,A -85,B 0,C 180,E1 -19223.712,E2 -19223.712} C_VEL
LIN {X 0,Y 243.579,Z 378.873,A -85,B 0,C 180,E1 -19226.798,E2 -19226.798} C_VEL
LIN {X 0,Y 243.043,Z 375.89,A -85,B 0,C 180,E1 -19230.556,E2 -19230.556} C_VEL
LIN {X 0,Y 242.548,Z 373.268,A -85,B 0,C 180,E1 -19234.238,E2 -19234.238} C_VEL
LIN {X 0,Y 242.055,Z 370.955,A -85,B 0,C 180,E1 -19238.297,E2 -19238.297} C_VEL
LIN {X 0,Y 242.165,Z 370.94,A -85,B 0,C 180,E1 -19243.279,E2 -19243.279} C_VEL
LIN {X 0,Y 242.184,Z 370.941,A -85,B 0,C 180,E1 -19248.28,E2 -19248.28} C_VEL
LIN {X 0,Y 242.397,Z 370.916,A -85,B 0,C 180,E1 -19251.665,E2 -19251.665} C_VEL
LIN {X 0,Y 242.259,Z 370.933,A -85,B 0,C 180,E1 -19255.007,E2 -19255.007} C_VEL
LIN {X 0,Y 242.639,Z 370.884,A -85,B 0,C 180,E1 -19258.341,E2 -19258.341} C_VEL
LIN {X 0,Y 242.639,Z 370.881,A -85,B 0,C 180,E1 -19261.66,E2 -19261.66} C_VEL
LIN {X 0,Y 242.432,Z 370.908,A -85,B 0,C 180,E1 -19266.753,E2 -19266.753} C_VEL
LIN {X 0,Y 242.348,Z 370.922,A -85,B 0,C 180,E1 -19270.021,E2 -19270.021} C_VEL
LIN {X 0,Y 242.17,Z 370.937,A -85,B 0,C 180,E1 -19275.141,E2 -19275.141} C_VEL
LIN {X 0,Y 242.077,Z 370.95,A -85,B 0,C 180,E1 -19278.624,E2 -19278.624} C_VEL
LIN {X 0,Y 242.016,Z 370.961,A -85,B 0,C 180,E1 -19282.18,E2 -19282.18} C_VEL
LIN {X 0,Y 242.069,Z 370.956,A -85,B 0,C 180,E1 -19285.838,E2 -19285.838} C_VEL
LIN {X 0,Y 242.033,Z 371.09,A -85,B 0,C 180,E1 -19289.58,E2 -19289.58} C_VEL
LIN {X 0,Y 242.406,Z 373.156,A -85,B 0,C 180,E1 -19293.426,E2 -19293.426} C_VEL
LIN {X 0,Y 242.856,Z 375.558,A -85,B 0,C 180,E1 -19297.425,E2 -19297.425} C_VEL
LIN {X 0,Y 243.275,Z 378.387,A -85,B 0,C 180,E1 -19301.641,E2 -19301.641} C_VEL
LIN {X 0,Y 243.536,Z 379.964,A -85,B 0,C 180,E1 -19303.837,E2 -19303.837} C_VEL
LIN {X 0,Y 243.78,Z 381.772,A -85,B 0,C 180,E1 -19306.219,E2 -19306.219} C_VEL
LIN {X 0,Y 243.971,Z 385.001,A -85,B 0,C 180,E1 -19309.983,E2 -19309.983} C_VEL
LIN {X 0,Y 245.141,Z 388.026,A -85,B 0,C 180,E1 -19310.358,E2 -19310.358} C_VEL
LIN {X 0,Y 246.487,Z 390.339,A -85,B 0,C 180,E1 -19310.731,E2 -19310.731} C_VEL
LIN {X 0,Y 251.356,Z 400.823,A -85,B 0,C 180,E1 -19312.276,E2 -19312.276} C_VEL
LIN {X 0,Y 255.546,Z 412.082,A -85,B 0,C 180,E1 -19313.889,E2 -19313.889} C_VEL
LIN {X 0,Y 259.185,Z 425.145,A -85,B 0,C 180,E1 -19315.794,E2 -19315.794} C_VEL
LIN {X 0,Y 261.362,Z 435.972,A -85,B 0,C 180,E1 -19317.466,E2 -19317.466} C_VEL
LIN {X 0,Y 262.548,Z 445.061,A -85,B 0,C 180,E1 -19318.936,E2 -19318.936} C_VEL
LIN {X 0,Y 262.595,Z 446.608,A -85,B 0,C 180,E1 -19319.189,E2 -19319.189} C_VEL
LIN {X 0,Y 259.751,Z 458.484,A -85,B 0,C 180,E1 -19320.855,E2 -19320.855} C_VEL
LIN {X 0,Y 256.693,Z 469.253,A -85,B 0,C 180,E1 -19322.703,E2 -19322.703} C_VEL
LIN {X 0,Y 253.536,Z 479.922,A -85,B 0,C 180,E1 -19324.993,E2 -19324.993} C_VEL
LIN {X 0,Y 250.56,Z 488.773,A -85,B 0,C 180,E1 -19327.314,E2 -19327.314} C_VEL
LIN {X 0,Y 248.253,Z 495.806,A -85,B 0,C 180,E1 -19329.565,E2 -19329.565} C_VEL
LIN {X 0,Y 245.637,Z 503.272,A -85,B 0,C 180,E1 -19332.517,E2 -19332.517} C_VEL
LIN {X 0,Y 243.433,Z 509.684,A -85,B 0,C 180,E1 -19335.795,E2 -19335.795} C_VEL
LIN {X 0,Y 241.847,Z 514.529,A -85,B 0,C 180,E1 -19339.112,E2 -19339.112} C_VEL
LIN {X 0,Y 241.105,Z 517.261,A -85,B 0,C 180,E1 -19341.62,E2 -19341.62} C_VEL
LIN {X 0,Y 240.444,Z 519.717,A -85,B 0,C 180,E1 -19344.97,E2 -19344.97} C_VEL
LIN {X 0,Y 240.1,Z 520.94,A -85,B 0,C 180,E1 -19348.323,E2 -19348.323} C_VEL
LIN {X 0,Y 240.1,Z 520.96,A -85,B 0,C 180,E1 -19351.678,E2 -19351.678} C_VEL
LIN {X 0,Y 240.432,Z 519.783,A -85,B 0,C 180,E1 -19355.031,E2 -19355.031} C_VEL
LIN {X 0,Y 241.046,Z 517.376,A -85,B 0,C 180,E1 -19358.383,E2 -19358.383} C_VEL
LIN {X 0,Y 242.171,Z 513.652,A -85,B 0,C 180,E1 -19361.721,E2 -19361.721} C_VEL
LIN {X 0,Y 243.876,Z 508.487,A -85,B 0,C 180,E1 -19365.032,E2 -19365.032} C_VEL
LIN {X 0,Y 245.597,Z 503.539,A -85,B 0,C 180,E1 -19367.486,E2 -19367.486} C_VEL
LIN {X 0,Y 248.211,Z 496.214,A -85,B 0,C 180,E1 -19370.406,E2 -19370.406} C_VEL
LIN {X 0,Y 250.455,Z 489.168,A -85,B 0,C 180,E1 -19372.696,E2 -19372.696} C_VEL
LIN {X 0,Y 253.428,Z 480.398,A -85,B 0,C 180,E1 -19375.019,E2 -19375.019} C_VEL
LIN {X 0,Y 256.603,Z 469.818,A -85,B 0,C 180,E1 -19377.307,E2 -19377.307} C_VEL
LIN {X 0,Y 259.669,Z 459.158,A -85,B 0,C 180,E1 -19379.155,E2 -19379.155} C_VEL
LIN {X 0,Y 262.55,Z 447.253,A -85,B 0,C 180,E1 -19380.846,E2 -19380.846} C_VEL
LIN {X 0,Y 262.492,Z 443.987,A -85,B 0,C 180,E1 -19381.37,E2 -19381.37} C_VEL
LIN {X 0,Y 260.695,Z 431.877,A -85,B 0,C 180,E1 -19383.309,E2 -19383.309} C_VEL
LIN {X 0,Y 257.842,Z 419.651,A -85,B 0,C 180,E1 -19385.143,E2 -19385.143} C_VEL
LIN {X 0,Y 253.674,Z 406.663,A -85,B 0,C 180,E1 -19387.022,E2 -19387.022} C_VEL
LIN {X 0,Y 248.931,Z 395.365,A -85,B 0,C 180,E1 -19388.664,E2 -19388.664} C_VEL
LIN {X 0,Y 247.41,Z 392.275,A -85,B 0,C 180,E1 -19389.14,E2 -19389.14} C_VEL
LIN {X 0,Y 245.669,Z 388.814,A -85,B 0,C 180,E1 -19389.648,E2 -19389.648} C_VEL
LIN {X 0,Y 244.127,Z 385.643,A -85,B 0,C 180,E1 -19390.105,E2 -19390.105} C_VEL
LIN {X 0,Y 243.954,Z 384.815,A -85,B 0,C 180,E1 -19390.232,E2 -19390.232} C_VEL
LIN {X 0,Y 243.773,Z 381.82,A -85,B 0,C 180,E1 -19393.883,E2 -19393.883} C_VEL
LIN {X 0,Y 243.561,Z 380.104,A -85,B 0,C 180,E1 -19396.169,E2 -19396.169} C_VEL
LIN {X 0,Y 243.041,Z 377.04,A -85,B 0,C 180,E1 -19400.493,E2 -19400.493} C_VEL
LIN {X 0,Y 242.67,Z 374.421,A -85,B 0,C 180,E1 -19404.604,E2 -19404.604} C_VEL
LIN {X 0,Y 242.223,Z 372.192,A -85,B 0,C 180,E1 -19408.516,E2 -19408.516} C_VEL
LIN {X 0,Y 242.067,Z 370.956,A -85,B 0,C 180,E1 -19411.026,E2 -19411.026} C_VEL
LIN {X 0,Y 242.071,Z 370.953,A -85,B 0,C 180,E1 -19414.183,E2 -19414.183} C_VEL
LIN {X 0,Y 242.057,Z 370.956,A -85,B 0,C 180,E1 -19418.297,E2 -19418.297} C_VEL
LIN {X 0,Y 242.167,Z 370.945,A -85,B 0,C 180,E1 -19423.278,E2 -19423.278} C_VEL
LIN {X 0,Y 242.191,Z 370.935,A -85,B 0,C 180,E1 -19428.28,E2 -19428.28} C_VEL
LIN {X 0,Y 242.44,Z 370.903,A -85,B 0,C 180,E1 -19431.666,E2 -19431.666} C_VEL
LIN {X 0,Y 242.265,Z 370.925,A -85,B 0,C 180,E1 -19435.007,E2 -19435.007} C_VEL
LIN {X 0,Y 242.641,Z 370.878,A -85,B 0,C 180,E1 -19438.34,E2 -19438.34} C_VEL
LIN {X 0,Y 242.64,Z 370.878,A -85,B 0,C 180,E1 -19441.659,E2 -19441.659} C_VEL
LIN {X 0,Y 242.421,Z 370.914,A -85,B 0,C 180,E1 -19446.659,E2 -19446.659} C_VEL
LIN {X 0,Y 242.271,Z 370.932,A -85,B 0,C 180,E1 -19450.023,E2 -19450.023} C_VEL
LIN {X 0,Y 242.171,Z 370.948,A -85,B 0,C 180,E1 -19455.14,E2 -19455.14} C_VEL
LIN {X 0,Y 242.083,Z 370.962,A -85,B 0,C 180,E1 -19458.623,E2 -19458.623} C_VEL
LIN {X 0,Y 242.073,Z 371.168,A -85,B 0,C 180,E1 -19462.174,E2 -19462.174} C_VEL
LIN {X 0,Y 242.601,Z 373.564,A -85,B 0,C 180,E1 -19466.095,E2 -19466.095} C_VEL
LIN {X 0,Y 243.102,Z 376.28,A -85,B 0,C 180,E1 -19469.854,E2 -19469.854} C_VEL
LIN {X 0,Y 243.591,Z 378.993,A -85,B 0,C 180,E1 -19473.242,E2 -19473.242} C_VEL
LIN {X 0,Y 244.206,Z 382.084,A -85,B 0,C 180,E1 -19476.77,E2 -19476.77} C_VEL
LIN {X 0,Y 243.778,Z 383.501,A -85,B 0,C 180,E1 -19478.112,E2 -19478.112} C_VEL
LIN {X 0,Y 241.417,Z 386.287,A -85,B 0,C 180,E1 -19480.29,E2 -19480.29} C_VEL
LIN {X 0,Y 239.411,Z 388.61,A -85,B 0,C 180,E1 -19482.055,E2 -19482.055} C_VEL
LIN {X 0,Y 238.662,Z 390.232,A -85,B 0,C 180,E1 -19483.422,E2 -19483.422} C_VEL
LIN {X 0,Y 238.664,Z 390.728,A -85,B 0,C 180,E1 -19483.886,E2 -19483.886} C_VEL
LIN {X 0,Y 239.095,Z 393.126,A -85,B 0,C 180,E1 -19486.142,E2 -19486.142} C_VEL
LIN {X 0,Y 240.421,Z 396.372,A -85,B 0,C 180,E1 -19486.571,E2 -19486.571} C_VEL
LIN {X 0,Y 241.851,Z 398.554,A -85,B 0,C 180,E1 -19486.978,E2 -19486.978} C_VEL
LIN {X 0,Y 244.078,Z 402.731,A -85,B 0,C 180,E1 -19487.639,E2 -19487.639} C_VEL
LIN {X 0,Y 249.252,Z 413.829,A -85,B 0,C 180,E1 -19489.363,E2 -19489.363} C_VEL
LIN {X 0,Y 251.652,Z 423.398,A -85,B 0,C 180,E1 -19490.566,E2 -19490.566} C_VEL
LIN {X 0,Y 253.755,Z 435.772,A -85,B 0,C 180,E1 -19492.16,E2 -19492.16} C_VEL
LIN {X 0,Y 255.131,Z 449.081,A -85,B 0,C 180,E1 -19494.006,E2 -19494.006} C_VEL
LIN {X 0,Y 255.473,Z 459.882,A -85,B 0,C 180,E1 -19495.618,E2 -19495.618} C_VEL
LIN {X 0,Y 255.155,Z 462.941,A -85,B 0,C 180,E1 -19496.074,E2 -19496.074} C_VEL
LIN {X 0,Y 251.6,Z 475.975,A -85,B 0,C 180,E1 -19497.945,E2 -19497.945} C_VEL
LIN {X 0,Y 248.402,Z 486.76,A -85,B 0,C 180,E1 -19499.854,E2 -19499.854} C_VEL
LIN {X 0,Y 244.982,Z 497.678,A -85,B 0,C 180,E1 -19502.213,E2 -19502.213} C_VEL
LIN {X 0,Y 241.709,Z 508.288,A -85,B 0,C 180,E1 -19505.064,E2 -19505.064} C_VEL
LIN {X 0,Y 238.764,Z 517.07,A -85,B 0,C 180,E1 -19507.957,E2 -19507.957} C_VEL
LIN {X 0,Y 236.559,Z 524.355,A -85,B 0,C 180,E1 -19510.925,E2 -19510.925} C_VEL
LIN {X 0,Y 234.703,Z 531.081,A -85,B 0,C 180,E1 -19514.365,E2 -19514.365} C_VEL
LIN {X 0,Y 233.457,Z 536.299,A -85,B 0,C 180,E1 -19517.835,E2 -19517.835} C_VEL
LIN {X 0,Y 232.927,Z 540.146,A -85,B 0,C 180,E1 -19521.323,E2 -19521.323} C_VEL
LIN {X 0,Y 232.838,Z 542.745,A -85,B 0,C 180,E1 -19524.919,E2 -19524.919} C_VEL
LIN {X 0,Y 232.917,Z 543.966,A -85,B 0,C 180,E1 -19528.271,E2 -19528.271} C_VEL
LIN {X 0,Y 232.948,Z 544.129,A -85,B 0,C 180,E1 -19530,E2 -19530} C_VEL
LIN {X 0,Y 232.918,Z 543.962,A -85,B 0,C 180,E1 -19531.729,E2 -19531.729} C_VEL
LIN {X 0,Y 232.839,Z 542.668,A -85,B 0,C 180,E1 -19535.195,E2 -19535.195} C_VEL
LIN {X 0,Y 232.927,Z 540.111,A -85,B 0,C 180,E1 -19538.677,E2 -19538.677} C_VEL
LIN {X 0,Y 233.456,Z 536.256,A -85,B 0,C 180,E1 -19542.165,E2 -19542.165} C_VEL
LIN {X 0,Y 234.663,Z 531.02,A -85,B 0,C 180,E1 -19545.637,E2 -19545.637} C_VEL
LIN {X 0,Y 236.557,Z 524.272,A -85,B 0,C 180,E1 -19549.075,E2 -19549.075} C_VEL
LIN {X 0,Y 238.752,Z 516.967,A -85,B 0,C 180,E1 -19552.044,E2 -19552.044} C_VEL
LIN {X 0,Y 241.654,Z 508.165,A -85,B 0,C 180,E1 -19554.942,E2 -19554.942} C_VEL
LIN {X 0,Y 244.966,Z 497.532,A -85,B 0,C 180,E1 -19557.788,E2 -19557.788} C_VEL
LIN {X 0,Y 248.375,Z 486.588,A -85,B 0,C 180,E1 -19560.149,E2 -19560.149} C_VEL
LIN {X 0,Y 251.926,Z 474.596,A -85,B 0,C 180,E1 -19562.245,E2 -19562.245} C_VEL
LIN {X 0,Y 255.131,Z 462.871,A -85,B 0,C 180,E1 -19563.899,E2 -19563.899} C_VEL
LIN {X 0,Y 255.432,Z 459.729,A -85,B 0,C 180,E1 -19564.369,E2 -19564.369} C_VEL
LIN {X 0,Y 254.892,Z 446.481,A -85,B 0,C 180,E1 -19566.338,E2 -19566.338} C_VEL
LIN {X 0,Y 253.466,Z 434.175,A -85,B 0,C 180,E1 -19568.017,E2 -19568.017} C_VEL
LIN {X 0,Y 250.847,Z 419.945,A -85,B 0,C 180,E1 -19569.821,E2 -19569.821} C_VEL
LIN {X 0,Y 248.768,Z 412.707,A -85,B 0,C 180,E1 -19570.757,E2 -19570.757} C_VEL
LIN {X 0,Y 243.834,Z 402.349,A -85,B 0,C 180,E1 -19572.374,E2 -19572.374} C_VEL
LIN {X 0,Y 241.018,Z 397.281,A -85,B 0,C 180,E1 -19573.199,E2 -19573.199} C_VEL
LIN {X 0,Y 239.37,Z 394.062,A -85,B 0,C 180,E1 -19573.699,E2 -19573.699} C_VEL
LIN {X 0,Y 239.091,Z 393.038,A -85,B 0,C 180,E1 -19573.857,E2 -19573.857} C_VEL
LIN {X 0,Y 238.382,Z 389.27,A -85,B 0,C 180,E1 -19577.481,E2 -19577.481} C_VEL
LIN {X 0,Y 237.601,Z 385.273,A -85,B 0,C 180,E1 -19581.6,E2 -19581.6} C_VEL
LIN {X 0,Y 236.895,Z 381.668,A -85,B 0,C 180,E1 -19585.69,E2 -19585.69} C_VEL
LIN {X 0,Y 236.326,Z 378.506,A -85,B 0,C 180,E1 -19589.632,E2 -19589.632} C_VEL
LIN {X 0,Y 235.842,Z 375.806,A -85,B 0,C 180,E1 -19593.449,E2 -19593.449} C_VEL
LIN {X 0,Y 235.256,Z 373.134,A -85,B 0,C 180,E1 -19597.834,E2 -19597.834} C_VEL
LIN {X 0,Y 234.983,Z 371.838,A -85,B 0,C 180,E1 -19600.338,E2 -19600.338} C_VEL
LIN {X 0,Y 235.117,Z 371.815,A -85,B 0,C 180,E1 -19604.394,E2 -19604.394} C_VEL
LIN {X 0,Y 235.217,Z 371.804,A -85,B 0,C 180,E1 -19609.673,E2 -19609.673} C_VEL
LIN {X 0,Y 235.371,Z 371.784,A -85,B 0,C 180,E1 -19613.141,E2 -19613.141} C_VEL
LIN {X 0,Y 235.599,Z 371.76,A -85,B 0,C 180,E1 -19618.291,E2 -19618.291} C_VEL
LIN {X 0,Y 235.599,Z 371.758,A -85,B 0,C 180,E1 -19621.71,E2 -19621.71} C_VEL
LIN {X 0,Y 235.409,Z 371.782,A -85,B 0,C 180,E1 -19626.859,E2 -19626.859} C_VEL
LIN {X 0,Y 235.256,Z 371.802,A -85,B 0,C 180,E1 -19630.326,E2 -19630.326} C_VEL
LIN {X 0,Y 235.117,Z 371.817,A -85,B 0,C 180,E1 -19635.606,E2 -19635.606} C_VEL
LIN {X 0,Y 235.012,Z 371.833,A -85,B 0,C 180,E1 -19639.206,E2 -19639.206} C_VEL
LIN {X 0,Y 234.964,Z 371.843,A -85,B 0,C 180,E1 -19642.883,E2 -19642.883} C_VEL
LIN {X 0,Y 234.99,Z 371.863,A -85,B 0,C 180,E1 -19647.377,E2 -19647.377} C_VEL
LIN {X 0,Y 235.223,Z 373.375,A -85,B 0,C 180,E1 -19650.526,E2 -19650.526} C_VEL
LIN {X 0,Y 235.619,Z 375.524,A -85,B 0,C 180,E1 -19654.523,E2 -19654.523} C_VEL
LIN {X 0,Y 236.065,Z 378.041,A -85,B 0,C 180,E1 -19658.697,E2 -19658.697} C_VEL
LIN {X 0,Y 236.499,Z 381.034,A -85,B 0,C 180,E1 -19663.117,E2 -19663.117} C_VEL
LIN {X 0,Y 236.836,Z 383.874,A -85,B 0,C 180,E1 -19666.959,E2 -19666.959} C_VEL
LIN {X 0,Y 236.966,Z 385.091,A -85,B 0,C 180,E1 -19668.468,E2 -19668.468} C_VEL
LIN {X 0,Y 238.242,Z 388.313,A -85,B 0,C 180,E1 -19668.901,E2 -19668.901} C_VEL
LIN {X 0,Y 239.581,Z 390.228,A -85,B 0,C 180,E1 -19669.283,E2 -19669.283} C_VEL
LIN {X 0,Y 245.089,Z 401.802,A -85,B 0,C 180,E1 -19671.133,E2 -19671.133} C_VEL
LIN {X 0,Y 249.629,Z 414.17,A -85,B 0,C 180,E1 -19673.022,E2 -19673.022} C_VEL
LIN {X 0,Y 253.11,Z 426.924,A -85,B 0,C 180,E1 -19674.995,E2 -19674.995} C_VEL
LIN {X 0,Y 255.392,Z 439.194,A -85,B 0,C 180,E1 -19676.983,E2 -19676.983} C_VEL
LIN {X 0,Y 256.308,Z 447.543,A -85,B 0,C 180,E1 -19678.42,E2 -19678.42} C_VEL
LIN {X 0,Y 253.933,Z 457.824,A -85,B 0,C 180,E1 -19679.907,E2 -19679.907} C_VEL
LIN {X 0,Y 251.023,Z 467.713,A -85,B 0,C 180,E1 -19681.578,E2 -19681.578} C_VEL
LIN {X 0,Y 247.662,Z 478.699,A -85,B 0,C 180,E1 -19683.906,E2 -19683.906} C_VEL
LIN {X 0,Y 244.506,Z 487.812,A -85,B 0,C 180,E1 -19686.271,E2 -19686.271} C_VEL
LIN {X 0,Y 241.542,Z 496.337,A -85,B 0,C 180,E1 -19689.04,E2 -19689.04} C_VEL
LIN {X 0,Y 238.881,Z 503.626,A -85,B 0,C 180,E1 -19692.006,E2 -19692.006} C_VEL
LIN {X 0,Y 236.56,Z 510.034,A -85,B 0,C 180,E1 -19695.373,E2 -19695.373} C_VEL
LIN {X 0,Y 234.892,Z 514.875,A -85,B 0,C 180,E1 -19698.786,E2 -19698.786} C_VEL
LIN {X 0,Y 234.084,Z 517.607,A -85,B 0,C 180,E1 -19701.366,E2 -19701.366} C_VEL
LIN {X 0,Y 233.385,Z 520.062,A -85,B 0,C 180,E1 -19704.817,E2 -19704.817} C_VEL
LIN {X 0,Y 233.032,Z 521.284,A -85,B 0,C 180,E1 -19708.272,E2 -19708.272} C_VEL
LIN {X 0,Y 233.032,Z 521.305,A -85,B 0,C 180,E1 -19711.728,E2 -19711.728} C_VEL
LIN {X 0,Y 233.372,Z 520.128,A -85,B 0,C 180,E1 -19715.184,E2 -19715.184} C_VEL
LIN {X 0,Y 234.016,Z 517.721,A -85,B 0,C 180,E1 -19718.636,E2 -19718.636} C_VEL
LIN {X 0,Y 235.23,Z 513.998,A -85,B 0,C 180,E1 -19722.072,E2 -19722.072} C_VEL
LIN {X 0,Y 237.023,Z 508.837,A -85,B 0,C 180,E1 -19725.478,E2 -19725.478} C_VEL
LIN {X 0,Y 238.841,Z 503.89,A -85,B 0,C 180,E1 -19727.997,E2 -19727.997} C_VEL
LIN {X 0,Y 241.506,Z 496.724,A -85,B 0,C 180,E1 -19730.937,E2 -19730.937} C_VEL
LIN {X 0,Y 243.937,Z 489.535,A -85,B 0,C 180,E1 -19733.338,E2 -19733.338} C_VEL
LIN {X 0,Y 247.016,Z 480.778,A -85,B 0,C 180,E1 -19735.715,E2 -19735.715} C_VEL
LIN {X 0,Y 250.332,Z 470.216,A -85,B 0,C 180,E1 -19738.051,E2 -19738.051} C_VEL
LIN {X 0,Y 253.822,Z 458.463,A -85,B 0,C 180,E1 -19740.114,E2 -19740.114} C_VEL
LIN {X 0,Y 256.345,Z 448.241,A -85,B 0,C 180,E1 -19741.593,E2 -19741.593} C_VEL
LIN {X 0,Y 255.484,Z 439.548,A -85,B 0,C 180,E1 -19743.086,E2 -19743.086} C_VEL
LIN {X 0,Y 253.275,Z 427.393,A -85,B 0,C 180,E1 -19745.058,E2 -19745.058} C_VEL
LIN {X 0,Y 250.236,Z 416.007,A -85,B 0,C 180,E1 -19746.828,E2 -19746.828} C_VEL
LIN {X 0,Y 245.812,Z 403.614,A -85,B 0,C 180,E1 -19748.739,E2 -19748.739} C_VEL
LIN {X 0,Y 241.428,Z 393.798,A -85,B 0,C 180,E1 -19750.282,E2 -19750.282} C_VEL
LIN {X 0,Y 238.96,Z 389.312,A -85,B 0,C 180,E1 -19751.046,E2 -19751.046} C_VEL
LIN {X 0,Y 237.314,Z 386.36,A -85,B 0,C 180,E1 -19751.55,E2 -19751.55} C_VEL
LIN {X 0,Y 236.941,Z 385.036,A -85,B 0,C 180,E1 -19751.727,E2 -19751.727} C_VEL
LIN {X 0,Y 236.665,Z 382.181,A -85,B 0,C 180,E1 -19755.456,E2 -19755.456} C_VEL
LIN {X 0,Y 236.275,Z 379.598,A -85,B 0,C 180,E1 -19759.126,E2 -19759.126} C_VEL
LIN {X 0,Y 235.862,Z 376.776,A -85,B 0,C 180,E1 -19763.565,E2 -19763.565} C_VEL
LIN {X 0,Y 235.485,Z 374.512,A -85,B 0,C 180,E1 -19767.506,E2 -19767.506} C_VEL
